(* Logix 5000 project; controller LeakTestAuto vendor 1 type 14 code 226 rev 37.11; software revision 37.01; part 2 of 14 *)

ADD_ON_INSTRUCTION AOI_RobotPositions   (* revision 1.0 *)
VAR_OUTPUT
   LoadingNest : DINT; {access Read Only}
   Barcode : DINT; {access Read Only}
   TestingNest1 : DINT; {access Read Only}
   TestingNest2 : DINT; {access Read Only}
   PassChute : DINT; {access Read Only}
   FailChute : DINT; {access Read Only}
END_VAR

ROUTINE Logic   (* structured text *)
   LoadingNest := 0;
   Barcode := 1;
   TestingNest1 := 2;
   TestingNest2 := 3;
   PassChute := 4;
   FailChute := 5;
END_ROUTINE
END_ADD_ON_INSTRUCTION

ADD_ON_INSTRUCTION AOI_Sequencer_x64   (* revision 1.0 *)
VAR_IN_OUT
   SequenceStructure : udt_SequenceStructure_X64; {required}
END_VAR
VAR_INPUT
   inpNextStepInterlock : BOOL; {access Read Only, required}
   inpCyclePause : BOOL; {access Read Only, required}
   inpStepMode : BOOL; {access Read Only, required}
END_VAR
VAR
   FFLUDumpREAL : REAL; {access None}
   Seq_FFLU_Cycle : CONTROL := (LEN := 10); {access None}
   Seq_FFLU_Step : CONTROL := (LEN := 64); {access None}
   Seq_FFLU_StepHist : CONTROL := (LEN := 64); {access None}
   FFLUDumpINT : INT; {access None}
   AvgContol : CONTROL := (LEN := 10); {access None}
END_VAR

ROUTINE Logic   (* ladder *)
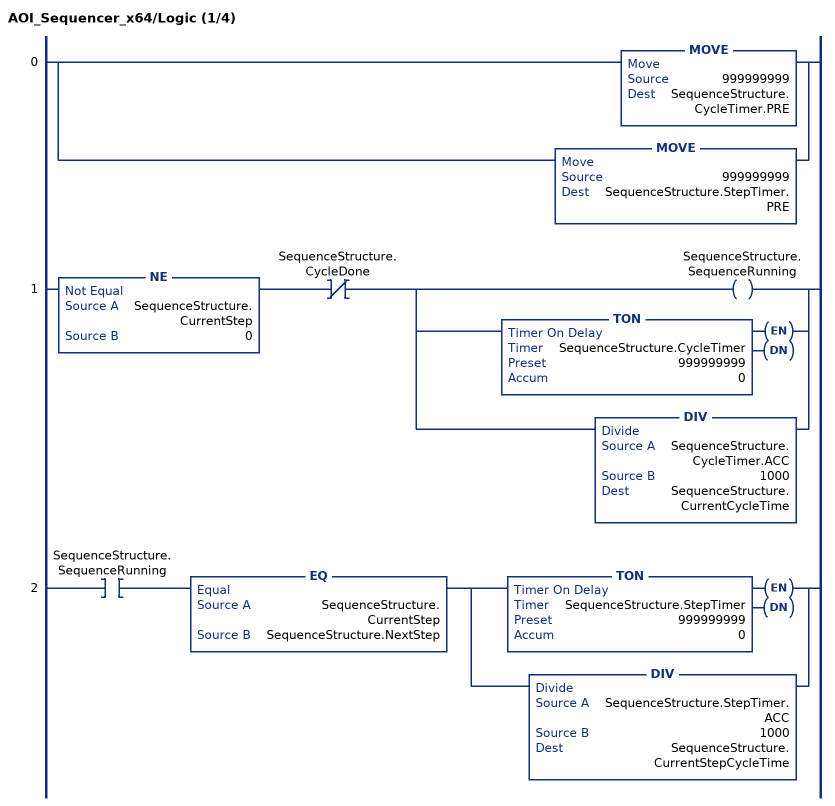
   0: [MOVE(999999999,SequenceStructure.CycleTimer.PRE) ,MOVE(999999999,SequenceStructure.StepTimer.PRE) ];
   1: NE(SequenceStructure.CurrentStep,0)XIO(SequenceStructure.CycleDone)[OTE(SequenceStructure.SequenceRunning) ,TON(SequenceStructure.CycleTimer,999999999,0) ,DIV(SequenceStructure.CycleTimer.ACC,1000,SequenceStructure.CurrentCycleTime) ];
   2: XIC(SequenceStructure.SequenceRunning)EQ(SequenceStructure.CurrentStep,SequenceStructure.NextStep)[TON(SequenceStructure.StepTimer,999999999,0) ,DIV(SequenceStructure.StepTimer.ACC,1000,SequenceStructure.CurrentStepCycleTime) ];
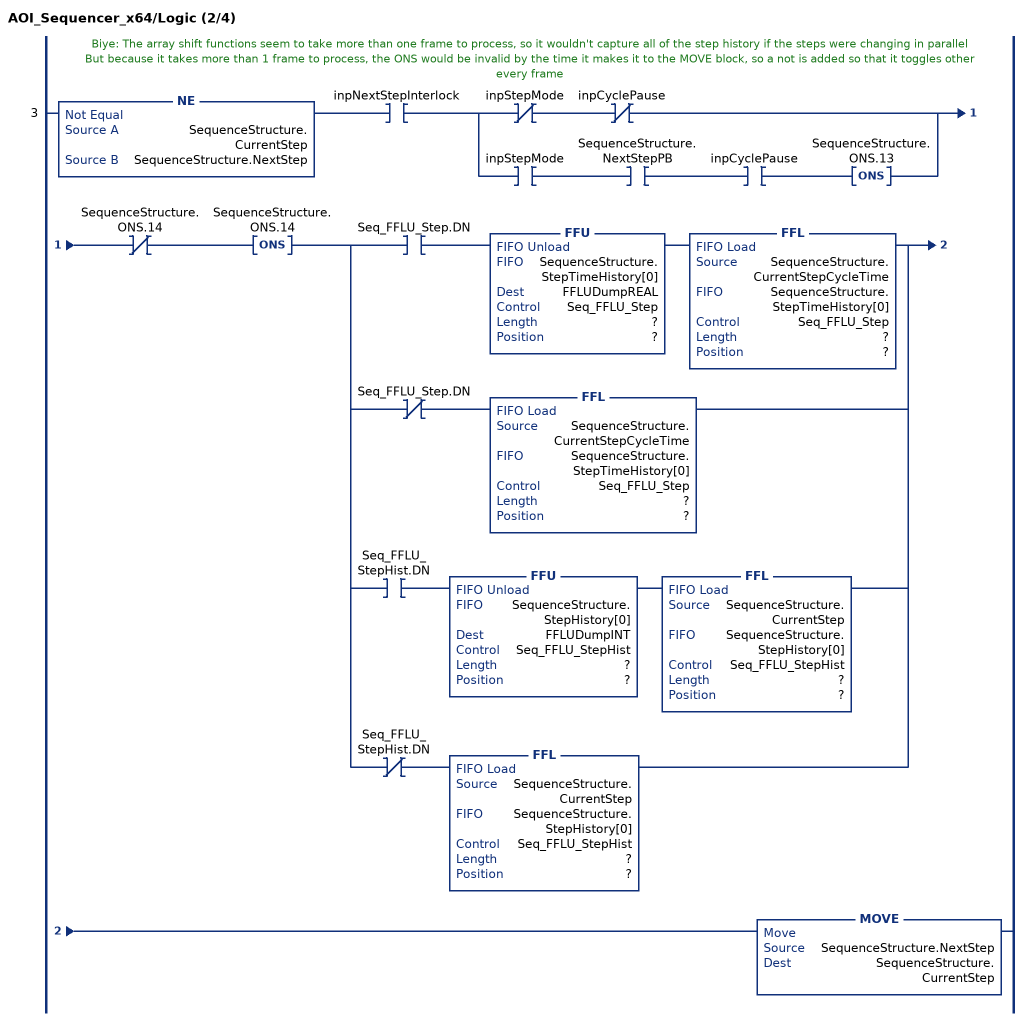
   // Biye: The array shift functions seem to take more than one frame to process, so it wouldn't capture all of the step history if the steps were changing in parallel
   // But because it takes more than 1 frame to process, the ONS would be invalid by the time it makes it to the MOVE block, so a not is added so that it toggles other every frame
   3: NE(SequenceStructure.CurrentStep,SequenceStructure.NextStep)XIC(inpNextStepInterlock)[XIO(inpStepMode) XIO(inpCyclePause) ,XIC(inpStepMode) XIC(SequenceStructure.NextStepPB) XIC(inpCyclePause) ONS(SequenceStructure.ONS.13) ]XIO(SequenceStructure.ONS.14)ONS(SequenceStructure.ONS.14)[XIC(Seq_FFLU_Step.DN) FFU(SequenceStructure.StepTimeHistory[0],FFLUDumpREAL,Seq_FFLU_Step,?,?) FFL(SequenceStructure.CurrentStepCycleTime,SequenceStructure.StepTimeHistory[0],Seq_FFLU_Step,?,?) ,XIO(Seq_FFLU_Step.DN) FFL(SequenceStructure.CurrentStepCycleTime,SequenceStructure.StepTimeHistory[0],Seq_FFLU_Step,?,?) ,XIC(Seq_FFLU_StepHist.DN) FFU(SequenceStructure.StepHistory[0],FFLUDumpINT,Seq_FFLU_StepHist,?,?) FFL(SequenceStructure.CurrentStep,SequenceStructure.StepHistory[0],Seq_FFLU_StepHist,?,?) ,XIO(Seq_FFLU_StepHist.DN) FFL(SequenceStructure.CurrentStep,SequenceStructure.StepHistory[0],Seq_FFLU_StepHist,?,?) ]MOVE(SequenceStructure.NextStep,SequenceStructure.CurrentStep);
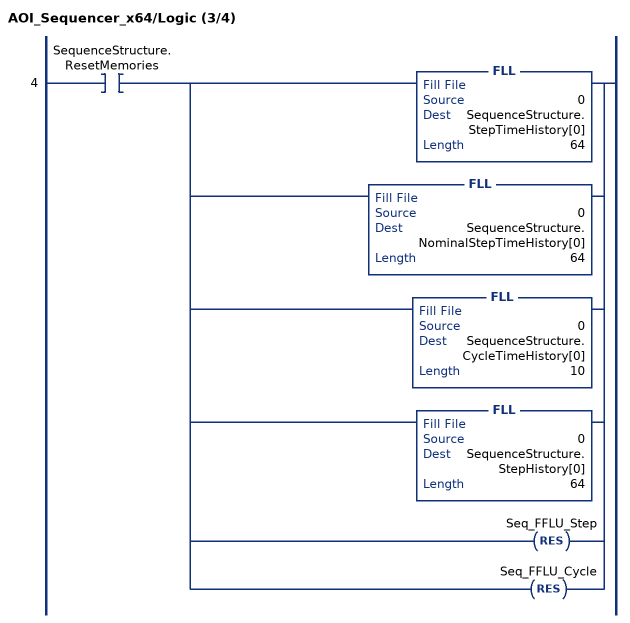
   4: XIC(SequenceStructure.ResetMemories)[FLL(0,SequenceStructure.StepTimeHistory[0],64) ,FLL(0,SequenceStructure.NominalStepTimeHistory[0],64) ,FLL(0,SequenceStructure.CycleTimeHistory[0],10) ,FLL(0,SequenceStructure.StepHistory[0],64) ,RES(Seq_FFLU_Step) ,RES(Seq_FFLU_Cycle) ];
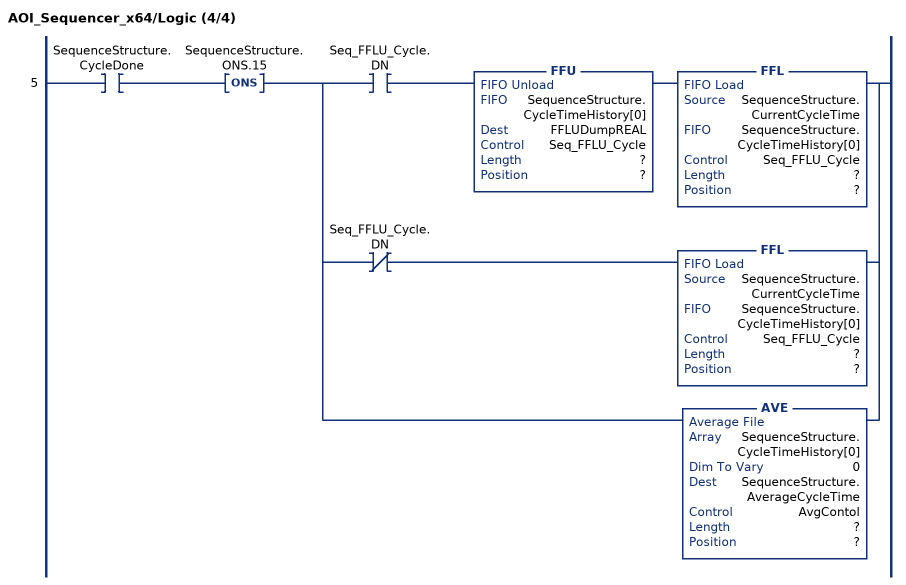
   5: XIC(SequenceStructure.CycleDone)ONS(SequenceStructure.ONS.15)[XIC(Seq_FFLU_Cycle.DN) FFU(SequenceStructure.CycleTimeHistory[0],FFLUDumpREAL,Seq_FFLU_Cycle,?,?) FFL(SequenceStructure.CurrentCycleTime,SequenceStructure.CycleTimeHistory[0],Seq_FFLU_Cycle,?,?) ,XIO(Seq_FFLU_Cycle.DN) FFL(SequenceStructure.CurrentCycleTime,SequenceStructure.CycleTimeHistory[0],Seq_FFLU_Cycle,?,?) ,AVE(SequenceStructure.CycleTimeHistory[0],0,SequenceStructure.AverageCycleTime,AvgContol,?,?) ];
END_ROUTINE
END_ADD_ON_INSTRUCTION

ADD_ON_INSTRUCTION AOI_StandardSeqSteps   (* revision 1.0 *)
VAR_OUTPUT
   Start : DINT; {access Read Only}
   ResultProcessing : DINT; {access Read Only}
   Complete : DINT; {access Read Only}
END_VAR

ROUTINE Logic   (* structured text *)
   Start := 1000;
   ResultProcessing := 8000;
   Complete := 9000;
END_ROUTINE
END_ADD_ON_INSTRUCTION

VAR_GLOBAL   (* controller tags *)
   AOI_IOCounter : AOI_IOCounter;
   ConveyorPurgeCounter : DINT;   // Outfeed Coveyor Purge Counter
   DateString : String20 := '07/14/2026';
   DateTimeString : String20 := '07/14/2026 13:25:59';
   Delay_TMR : TIMER[11] := ([0].PRE := 500, [1].PRE := 500, [3].PRE := 1000, [10].PRE := 100);   // Delay Timers
   HMI_ClearProcessFaultCounts_PB : BOOL;
   HMI_PurgeCycleSP : DINT := 20;   // HMI Purge Cycles Setpoint
   I_OP220_N3_CONVEYOR_CLEAT : ALIAS FOR Local:3:I.Pt13.Data;
   I_OP220_N3_CONVEYOR_LOAD : ALIAS FOR Local:3:I.Pt12.Data;
   I_OP220_N3_CONVEYOR_UNLOAD : ALIAS FOR Local:3:I.Pt14.Data;
   I_OP220_N3_DUT_PRE_NEST_0 : ALIAS FOR Local:3:I.Pt00.Data;
   I_OP220_N3_DUT_PRE_NEST_1 : ALIAS FOR Local:3:I.Pt01.Data;
   I_OP220_N3_DUT_PRE_NEST_2 : ALIAS FOR Local:3:I.Pt02.Data;
   I_OP220_N3_MAIN_AIR_OK : ALIAS FOR Local:3:I.Pt07.Data;
   I_OP220_N3_NEST1_EXTEND : ALIAS FOR Local:3:I.Pt04.Data;
   I_OP220_N3_NEST1_HOME : ALIAS FOR Local:3:I.Pt03.Data;
   I_OP220_N3_NEST2_EXTEND : ALIAS FOR Local:3:I.Pt06.Data;
   I_OP220_N3_NEST2_HOME : ALIAS FOR Local:3:I.Pt05.Data;
   I_OP220_N3_REJECT_BIN_OK : ALIAS FOR Local:3:I.Pt09.Data;
   I_OP220_N3_REJECT_CHUTE_PART : ALIAS FOR Local:3:I.Pt10.Data;
   I_OP220_N4_AC_SURGE_OK : ALIAS FOR Local:4:I.Pt00.Data;
   I_OP220_N4_CONVEYOR_ALARM_OK : ALIAS FOR Local:4:I.Pt03.Data;
   I_OP220_N4_CONVEYOR_SPEED : ALIAS FOR Local:4:I.Pt02.Data;
   I_OP220_N4_DC_OK : ALIAS FOR Local:4:I.Pt01.Data;
   I_OP220_N4_DC_OK_PS2 : ALIAS FOR Local:4:I.Pt04.Data;
   Ignition_Bypass : BOOL := 1;
   Ignition_DataReady : BOOL;
   Ignition_DataReceived : BOOL;
   IOCounterHasRef : BOOL := 1;
   IOCounterLastData : INT[8] := ([0] := 30383, [1] := 27, [2] := -31920);
   IOLabels : STRING[128] := ([0] := 'SI_OP220_N1_LASER_AREA_NC12', [1] := 'SI_OP220_N1_LASER_GUARD_NC12', [3] := 'SI_OP220_N1_SSR_12', [4] := 'SI_OP220_N1_CTRL_VLAVE_NC1', [8] := 'SO_OP220_N2_SSR_1', [9] := 'SO_OP220_N2_SSR_2', [16] := 'I_OP220_N3_DUT_PRE_NEST_0', [17] := 'I_OP220_N3_DUT_PRE_NEST_1', [18] := 'I_OP220_N3_DUT_PRE_NEST_2', [19] := 'I_OP220_N3_NEST1_HOME', [20] := 'I_OP220_N3_NEST1_EXTEND', [21] := 'I_OP220_N3_NEST2_HOME', [22] := 'I_OP220_N3_NEST2_EXTEND', [23] := 'I_OP220_N3_MAIN_AIR_OK', [25] := 'I_OP220_N3_REJECT_BIN_OK', [26] := 'I_OP220_N3_REJECT_CHUTE_PART', [28] := 'I_OP220_N3_CONVEYOR_LOAD', [29] := 'I_OP220_N3_CONVEYOR_CLEAT', [30] := 'I_OP220_N3_CONVEYOR_UNLOAD', [32] := 'I_OP220_N4_AC_SURGE_OK', [33] := 'I_OP220_N4_DC_OK', [34] := 'I_OP220_N4_CONVEYOR_SPEED', [35] := 'I_OP220_N4_CONVEYOR_ALARM_OK', [36] := 'I_OP220_N4_DC_OK_PS2', [48] := 'O_OP220_N5_EN_LT_GN', [49] := 'O_OP220_N5_EN_LT_YE', [50] := 'O_OP220_N5_EN_LT_RD', [51] := 'O_OP220_N5_EN_LT_BU', [52] := 'O_OP220_N5_EN_MAIN_AIR', [53] := 'O_OP220_N5_EN_NEST1_EXT', [54] := 'O_OP220_N5_EN_NEST1_HOME', [55] := 'O_OP220_N5_EN_NEST2_EXT', [56] := 'O_OP220_N5_EN_NEST2_HOME', [57] := 'O_OP220_N5_EN_ROBOT_LATCHOFF', [58] := 'O_OP220_N5_EN_CONV_ALM_RST', [59] := 'O_OP220_N5_CONV_REV', [60] := 'O_OP220_N5_CONV_FWD', [62] := 'O_OP220_N5_EN_GRIPPER_GRIP', [63] := 'O_OP220_N5_EN_GRIPPER_UNGRIP');
   IOResetArray : INT[8];
   IOTriggerCounts : UDINT[128] := ([0] := 204299, [1] := 372945, [2] := 289990, [3] := 273, [4] := 284, [5] := 267, [6] := 273, [7] := 59, [8] := 521, [9] := 265, [10] := 457, [11] := 1168, [12] := 461, [13] := 232, [14] := 218066, [16] := 969840, [17] := 969667, [18] := 22, [19] := 986, [21] := 84223, [22] := 84230, [23] := 72795, [24] := 72777, [25] := 484, [26] := 4412, [28] := 201946, [29] := 3, [30] := 359046, [31] := 359046);
   James_Dint : DINT := 27;   // James Test Word
   LastPLCEdit : String20 := '12/31/1997 20:30:57';
   LastPLCEditHistory : String20[20] := ([0] := '12/31/1997 20:30:57', [1] := '12/31/1997 20:25:04', [2] := '12/31/1997 20:25:02', [3] := '12/31/1997 20:23:56', [4] := '07/13/2026 19:08:25', [5] := '07/13/2026 19:08:18', [6] := '07/13/2026 19:08:11', [7] := '07/13/2026 19:08:03', [8] := '07/13/2026 19:07:56', [9] := '07/13/2026 19:07:30', [10] := '07/13/2026 19:07:23', [11] := '07/13/2026 19:07:15', [12] := '07/13/2026 19:07:07', [13] := '07/13/2026 19:06:54', [14] := '07/13/2026 18:39:24', [15] := '07/13/2026 18:31:47', [16] := '07/13/2026 18:28:19', [17] := '07/13/2026 18:25:40', [18] := '07/13/2026 18:21:57', [19] := '07/13/2026 18:19:53');
   NoData : AB:5000_DI16:I:0;
   null : STRING;
   O_OP220_N5_CONV_FWD : ALIAS FOR Local:5:O.Pt12.Data;
   O_OP220_N5_CONV_REV : ALIAS FOR Local:5:O.Pt11.Data;
   O_OP220_N5_EN_CONV_ALM_RST : ALIAS FOR Local:5:O.Pt10.Data;
   O_OP220_N5_EN_GRIPPER_GRIP : ALIAS FOR Local:5:O.Pt14.Data;
   O_OP220_N5_EN_GRIPPER_UNGRIP : ALIAS FOR Local:5:O.Pt15.Data;
   O_OP220_N5_EN_LT_BU : ALIAS FOR Local:5:O.Pt03.Data;
   O_OP220_N5_EN_LT_GN : ALIAS FOR Local:5:O.Pt00.Data;
   O_OP220_N5_EN_LT_RD : ALIAS FOR Local:5:O.Pt02.Data;
   O_OP220_N5_EN_LT_YE : ALIAS FOR Local:5:O.Pt01.Data;
   O_OP220_N5_EN_MAIN_AIR : ALIAS FOR Local:5:O.Pt04.Data;
   O_OP220_N5_EN_NEST1_EXT : ALIAS FOR Local:5:O.Pt05.Data;
   O_OP220_N5_EN_NEST1_HOME : ALIAS FOR Local:5:O.Pt06.Data;
   O_OP220_N5_EN_NEST2_EXT : ALIAS FOR Local:5:O.Pt07.Data;
   O_OP220_N5_EN_NEST2_HOME : ALIAS FOR Local:5:O.Pt08.Data;
   O_OP220_N5_EN_ROBOT_LATCHOFF : ALIAS FOR Local:5:O.Pt09.Data;
   Oneshot : DINT;   // Oneshots
   OP220_ConsumedFromMain : DINT[50] := ([0] := 2, [1] := 3);
   OP220_ConsumedFromMain_PurgeModeEn : BOOL;
   OP220_ConsumedFromMain_RobotPickupSafe : BOOL := 1;
   OP220_EStop_OK : BOOL := 1;
   OP220_EStopTest_DCS : DCI_STOP := (ChannelA := 1, ChannelB := 1, InputStatus := 1, RestartType := 1, ColdStartType := 1, DiscrepancyTime := 250, O1 := 1);
   OP220_Power : BOOL := 1;
   OP220_ProducedForMain : DINT[50] := ([0] := 3); {produced}
   PLC : AOI_PLC := (AlwaysOn := 1, FlasherSlow := 1, FlasherFast := 1, SlowFlashTime := 2000, MediumFlashTime := 1000, FastFlashTime := 500, Year := 2026, Day := 14, Month := 7, Hour := 13, Minute := 25, Second := 59, MicroSecond := 766719, DOY := 195, SetTimePB := 1);
   Produced_SetTime : udt_Produced_SetTime := (SetTime[0] := 2020, SetTime[1] := 5, SetTime[2] := 21, SetTime[3] := 15, SetTime[4] := 59, SetTime[5] := 15); {produced}
   Purge_Count_DN : BOOL;   // Purge Counter Completed
   ShiftChange : BOOL;
   ShiftNumber : SINT := 1;
   SI_OP220_N1_CTRL_VLAVE_NC1 : ALIAS FOR Local:1:I.Pt04.Data;
   SI_OP220_N1_LASER_AREA_NC12 : ALIAS FOR Local:1:I.Pt00.Data;
   SI_OP220_N1_LASER_GUARD_NC12 : ALIAS FOR Local:1:I.Pt01.Data;
   SI_OP220_N1_SSR_12 : ALIAS FOR Local:1:I.Pt03.Data;
   SO_OP220_N2_SSR_1 : ALIAS FOR Local:2:O.Pt00.Data;
   SO_OP220_N2_SSR_2 : ALIAS FOR Local:2:O.Pt01.Data;
   ST1_Ignition_DataReady : BOOL;
   ST1_Ignition_DataReady_Setup : BOOL;
   ST1_Ignition_DataReceived : BOOL;
   ST1_Ignition_SerialNum : STRING := 'B252620969';
   ST1_Ignition_Status : DINT := -10;
   ST2_Ignition_DataReady : BOOL;
   ST2_Ignition_DataReady_Setup : BOOL;
   ST2_Ignition_DataReceived : BOOL;
   ST2_Ignition_SerialNum : STRING;
   ST2_Ignition_Status : DINT := -10;
   TimeString : String20 := '13:25:59';
   TON_PLC_BootUp : TIMER := (PRE := 10000);
END_VAR

PROGRAM MainProgram   (* main routine MainRoutine *)
VAR
   AOI_Barcode_Comms : AOI_CommStatus := (Cmd := 1, stsConnecting := 1, stsRunning := 1, stsFaultCode := 516);
   AOI_CapActuators_Seq : AOI_Sequencer_x64 := (inpNextStepInterlock := 1);
   AOI_CapCTS_Seq : AOI_Sequencer_x64 := (inpNextStepInterlock := 1);
   AOI_CapCylinders_Seq : AOI_Sequencer_x64 := (inpNextStepInterlock := 1);
   AOI_CapFail_Seq : AOI_Sequencer_x64 := (inpNextStepInterlock := 1);
   AOI_CapPass_Seq : AOI_Sequencer_x64 := (inpNextStepInterlock := 1);
   AOI_CapRobot_Seq : AOI_Sequencer_x64 := (inpNextStepInterlock := 1);
   AOI_CapShuffle_Seq : AOI_Sequencer_x64 := (inpNextStepInterlock := 1);
   AOI_Conveyor_Seq : AOI_Sequencer_x64 := (inpNextStepInterlock := 1);
   AOI_CTS1 : AOI_CTS_INSTRUMENT := (Change_Program_Number := 3, UID_of_Desired_Results := 43055, Include_Detailed_Results := 1, Results_Error := 1, UID_Time := 1300);
   AOI_CTS1_Comms : AOI_CommStatus := (Cmd := 1, stsFaulted := 1, stsRunning := 1, stsFaultCode := 516);
   AOI_CTS1_Seq : AOI_Sequencer_x64 := (inpNextStepInterlock := 1);
   AOI_CTS2 : AOI_CTS_INSTRUMENT := (Change_Program_Number := 3, UID_of_Desired_Results := 42054, Include_Detailed_Results := 1, Results_Error := 1, UID_Time := 1300);
   AOI_CTS2_Comms : AOI_CommStatus := (Cmd := 1, stsFaulted := 1, stsRunning := 1, stsFaultCode := 516);
   AOI_CTS2_Seq : AOI_Sequencer_x64 := (inpNextStepInterlock := 1);
   AOI_GetShift : AOI_GetShift := (PLCHour := 13, ShiftNumber := 1);
   AOI_OP220_HomingSeq : AOI_Sequencer_x64;
   AOI_OP220_Seq : AOI_Sequencer_x64 := (inpNextStepInterlock := 1);
   AOI_Robot_Comms : AOI_CommStatus := (Cmd := 1, stsRunning := 1, stsFaultCode := 272);
   AOI_RobotPos : AOI_RobotPositions := (Barcode := 1, TestingNest1 := 2, TestingNest2 := 3, PassChute := 4, FailChute := 5);
   AOI_SeqSteps : AOI_StandardSeqSteps := (Start := 1000, ResultProcessing := 8000, Complete := 9000);
   AOI_SRX100 : AOI_KeyenceBarcode := (ReadSuccess := 1);
   Barcode_ResultData : STR_Barcode := 'B252620969';
   BarcodeBypass : BOOL;
   BarcodeInputs : udt_KeyenceScannerInputs;
   BarcodeOutputs : udt_KeyenceScannerOutputs;
   BarcodeScanner : udt_OutputStructure := (IL := 1);
   CapActuators_BarcodeBad : COUNTER := (PRE := 999999999, CU := 1);
   CapActuators_BarcodeGood : COUNTER := (PRE := 999999999, ACC := 111, CU := 1);
   CapActuators_CTS1Bad : COUNTER := (PRE := 999999999, CU := 1);
   CapActuators_CTS1Good : COUNTER := (PRE := 999999999, ACC := 10, CU := 1);
   CapActuators_CTS2Bad : COUNTER := (PRE := 999999999, CU := 1);
   CapActuators_CTS2Good : COUNTER := (PRE := 999999999, ACC := 3, CU := 1);
   CapActuators_Nest1HasPart : BOOL := 1;
   CapActuators_Nest2HasPart : BOOL;
   CapActuators_Seq : udt_SequenceStructure_X64 := (ONS := -7937, CurrentCycleTime := 409000.0, StepTimer.PRE := 999999999, CycleTimer.PRE := 999999999);
   CapCTS_CTS1Bad : COUNTER := (PRE := 999999999, ACC := 356, CU := 1);
   CapCTS_CTS1Good : COUNTER := (PRE := 999999999, ACC := 2730, CU := 1);
   CapCTS_CTS2Bad : COUNTER := (PRE := 999999999, ACC := 1, CU := 1);
   CapCTS_CTS2Good : COUNTER := (PRE := 999999999, ACC := 3085, CU := 1);
   CapCTS_Nest1HasPart : BOOL := 1;
   CapCTS_Nest2HasPart : BOOL := 1;
   CapCTS_Seq : udt_SequenceStructure_X64 := (ONS := -8132, StepHistory[0] := 2000, StepHistory[1] := 2010, StepHistory[2] := 2000, StepHistory[3] := 2010, StepHistory[4] := 2000, StepHistory[5] := 2010, StepHistory[6] := 2000, StepHistory[7] := 2010, StepHistory[8] := 2000, StepHistory[9] := 2010, StepHistory[10] := 2000, StepHistory[11] := 2010, StepHistory[12] := 2000, StepHistory[13] := 2010, StepHistory[14] := 2000, StepHistory[15] := 2010, StepHistory[16] := 2000, StepHistory[17] := 2010, StepHistory[18] := 2000, StepHistory[19] := 2010, StepHistory[20] := 2000, StepHistory[21] := 2010, StepHistory[22] := 2000, StepHistory[23] := 2010, StepHistory[24] := 2000, StepHistory[25] := 2010, StepHistory[26] := 2000, StepHistory[27] := 2010, StepHistory[28] := 2000, StepHistory[29] := 2010, StepHistory[30] := 2000, StepHistory[31] := 2010, StepHistory[32] := 2000, StepHistory[33] := 2010, StepHistory[34] := 2000, StepHistory[35] := 2010, StepHistory[36] := 2000, StepHistory[37] := 2010, StepHistory[38] := 2000, StepHistory[39] := 2010, StepHistory[40] := 2000, StepHistory[41] := 2010, StepHistory[42] := 2000, StepHistory[43] := 2010, StepHistory[44] := 2000, StepHistory[45] := 2010, StepHistory[46] := 2000, StepHistory[47] := 2010, StepHistory[48] := 2000, StepHistory[49] := 2010, StepHistory[50] := 2000, StepHistory[51] := 2010, StepHistory[52] := 2000, StepHistory[53] := 2010, StepHistory[54] := 2000, StepHistory[55] := 2010, StepHistory[56] := 2000, StepHistory[57] := 2010, StepHistory[58] := 2000,
        StepHistory[59] := 2010, StepHistory[60] := 2000, StepHistory[61] := 2010, StepHistory[62] := 2000, StepHistory[63] := 2010, CurrentCycleTime := 66060.766, CurrentStepCycleTime := 387.139, StepTimeHistory[0] := 0.035, StepTimeHistory[1] := 21.3, StepTimeHistory[2] := 0.04, StepTimeHistory[3] := 21.295, StepTimeHistory[4] := 0.035, StepTimeHistory[5] := 21.266, StepTimeHistory[6] := 0.034, StepTimeHistory[7] := 21.271, StepTimeHistory[8] := 0.033, StepTimeHistory[9] := 21.285, StepTimeHistory[10] := 0.041, StepTimeHistory[11] := 21.294, StepTimeHistory[12] := 0.052, StepTimeHistory[13] := 21.304, StepTimeHistory[14] := 0.035, StepTimeHistory[15] := 21.297, StepTimeHistory[16] := 0.036, StepTimeHistory[17] := 21.266, StepTimeHistory[18] := 0.039, StepTimeHistory[19] := 21.292, StepTimeHistory[20] := 0.04, StepTimeHistory[21] := 21.273, StepTimeHistory[22] := 0.035, StepTimeHistory[23] := 21.271, StepTimeHistory[24] := 0.051, StepTimeHistory[25] := 21.29, StepTimeHistory[26] := 0.036, StepTimeHistory[27] := 21.274, StepTimeHistory[28] := 0.041, StepTimeHistory[29] := 21.289, StepTimeHistory[30] := 0.036, StepTimeHistory[31] := 21.285, StepTimeHistory[32] := 0.039, StepTimeHistory[33] := 21.296, StepTimeHistory[34] := 0.05, StepTimeHistory[35] := 21.273, StepTimeHistory[36] := 0.057, StepTimeHistory[37] := 21.274, StepTimeHistory[38] := 0.034, StepTimeHistory[39] := 21.285, StepTimeHistory[40] := 0.05, StepTimeHistory[41] := 21.27, StepTimeHistory[42] := 0.036, StepTimeHistory[43] := 21.29, StepTimeHistory[44] := 0.035, StepTimeHistory[45] := 21.309, StepTimeHistory[46] := 0.051, StepTimeHistory[47] := 21.274, StepTimeHistory[48] := 0.037, StepTimeHistory[49] := 21.315, StepTimeHistory[50] := 0.044, StepTimeHistory[51] := 21.296, StepTimeHistory[52] := 0.035,
        StepTimeHistory[53] := 21.271, StepTimeHistory[54] := 0.034, StepTimeHistory[55] := 21.289, StepTimeHistory[56] := 0.045, StepTimeHistory[57] := 21.29, StepTimeHistory[58] := 0.034, StepTimeHistory[59] := 21.296, StepTimeHistory[60] := 0.035, StepTimeHistory[61] := 21.293, StepTimeHistory[62] := 0.069, StepTimeHistory[63] := 21.691, StepTimer.PRE := 999999999, CycleTimer.PRE := 999999999);
   CapCylinders_Seq : udt_SequenceStructure_X64 := (ONS := -8192);
   CapFail_Seq : udt_SequenceStructure_X64 := (ONS := -8192);
   CapPass_Seq : udt_SequenceStructure_X64 := (ONS := -8191);
   CapRobot_IsNest : BOOL;
   CapRobot_Seq : udt_SequenceStructure_X64 := (ONS := -8191, StepHistory[0] := 2070, StepHistory[1] := 2000, StepHistory[2] := 2010, StepHistory[3] := 2020, StepHistory[4] := 2030, StepHistory[5] := 2050, StepHistory[6] := 2060, StepHistory[7] := 2070, StepHistory[8] := 2000, StepHistory[9] := 2010, StepHistory[10] := 2020, StepHistory[11] := 2030, StepHistory[12] := 2040, StepHistory[13] := 2050, StepHistory[14] := 2060, StepHistory[15] := 2070, StepHistory[16] := 2000, StepHistory[17] := 2010, StepHistory[18] := 2020, StepHistory[19] := 2030, StepHistory[20] := 2040, StepHistory[21] := 2050, StepHistory[22] := 2060, StepHistory[23] := 2070, StepHistory[24] := 2000, StepHistory[25] := 2010, StepHistory[26] := 2020, StepHistory[27] := 2030, StepHistory[28] := 2050, StepHistory[29] := 2060, StepHistory[30] := 2070, StepHistory[31] := 2000, StepHistory[32] := 2010, StepHistory[33] := 2020, StepHistory[34] := 2030, StepHistory[35] := 2050, StepHistory[36] := 2060, StepHistory[37] := 2070, StepHistory[38] := 2000, StepHistory[39] := 2010, StepHistory[40] := 2020, StepHistory[41] := 2030, StepHistory[42] := 2040, StepHistory[43] := 2050, StepHistory[44] := 2060, StepHistory[45] := 2070, StepHistory[46] := 2000, StepHistory[47] := 2010, StepHistory[48] := 2020, StepHistory[49] := 2030, StepHistory[50] := 2040, StepHistory[51] := 2050, StepHistory[52] := 2060, StepHistory[53] := 2070, StepHistory[54] := 2000, StepHistory[55] := 2010, StepHistory[56] := 2020, StepHistory[57] := 2030, StepHistory[58] := 2050,
        StepHistory[59] := 2060, StepHistory[60] := 2070, StepHistory[61] := 2000, StepHistory[62] := 2010, StepHistory[63] := 2020, CurrentCycleTime := 1115.231, CurrentStepCycleTime := 0.264, StepTimeHistory[0] := 0.789, StepTimeHistory[1] := 0.038, StepTimeHistory[2] := 1.379, StepTimeHistory[3] := 0.038, StepTimeHistory[4] := 0.759, StepTimeHistory[5] := 0.039, StepTimeHistory[6] := 0.908, StepTimeHistory[7] := 0.908, StepTimeHistory[8] := 0.908, StepTimeHistory[9] := 0.097, StepTimeHistory[10] := 0.039, StepTimeHistory[11] := 0.899, StepTimeHistory[12] := 0.089, StepTimeHistory[13] := 0.028, StepTimeHistory[14] := 0.909, StepTimeHistory[15] := 0.909, StepTimeHistory[16] := 0.909, StepTimeHistory[17] := 0.087, StepTimeHistory[18] := 0.029, StepTimeHistory[19] := 1.589, StepTimeHistory[20] := 0.099, StepTimeHistory[21] := 0.039, StepTimeHistory[22] := 1.559, StepTimeHistory[23] := 1.559, StepTimeHistory[24] := 1.559, StepTimeHistory[25] := 0.097, StepTimeHistory[26] := 0.029, StepTimeHistory[27] := 1.398, StepTimeHistory[28] := 0.038, StepTimeHistory[29] := 1.468, StepTimeHistory[30] := 1.468, StepTimeHistory[31] := 1.468, StepTimeHistory[32] := 0.088, StepTimeHistory[33] := 0.028, StepTimeHistory[34] := 1.279, StepTimeHistory[35] := 0.039, StepTimeHistory[36] := 1.399, StepTimeHistory[37] := 1.399, StepTimeHistory[38] := 0.028, StepTimeHistory[39] := 0.769, StepTimeHistory[40] := 0.029, StepTimeHistory[41] := 0.758, StepTimeHistory[42] := 0.009, StepTimeHistory[43] := 0.039, StepTimeHistory[44] := 0.66, StepTimeHistory[45] := 0.66, StepTimeHistory[46] := 0.66, StepTimeHistory[47] := 0.66, StepTimeHistory[48] := 0.037, StepTimeHistory[49] := 1.209, StepTimeHistory[50] := 0.099, StepTimeHistory[51] := 0.028, StepTimeHistory[52] := 1.049,
        StepTimeHistory[53] := 1.049, StepTimeHistory[54] := 1.049, StepTimeHistory[55] := 1.049, StepTimeHistory[56] := 0.036, StepTimeHistory[57] := 0.898, StepTimeHistory[58] := 0.038, StepTimeHistory[59] := 0.849, StepTimeHistory[60] := 0.849, StepTimeHistory[61] := 0.849, StepTimeHistory[62] := 0.849, StepTimeHistory[63] := 0.026, StepTimer.PRE := 999999999, CycleTimer.PRE := 999999999);
   CapRobot_StartPos : DINT := 1;
   CapRobot_TargetPos : DINT := 5;
   CapShuffle_CTS1Bad : COUNTER := (PRE := 999999999, ACC := 4, CU := 1);
   CapShuffle_CTS1Good : COUNTER := (PRE := 999999999, CU := 1);
   CapShuffle_CTS2Bad : COUNTER := (PRE := 999999999, ACC := 3, CU := 1);
   CapShuffle_CTS2Good : COUNTER := (PRE := 999999999, CU := 1);
   CapShuffle_Seq : udt_SequenceStructure_X64 := (ONS := -8161, StepHistory[0] := 5440, StepHistory[1] := 5450, StepHistory[2] := 4000, StepHistory[3] := 4010, StepHistory[4] := 4020, StepHistory[5] := 5000, StepHistory[6] := 5600, StepHistory[7] := 5610, StepHistory[8] := 5620, StepHistory[9] := 5630, StepHistory[10] := 5640, StepHistory[11] := 5650, StepHistory[12] := 4000, StepHistory[13] := 4010, StepHistory[14] := 4020, StepHistory[15] := 4030, StepHistory[16] := 5000, StepHistory[17] := 5100, StepHistory[18] := 5110, StepHistory[19] := 5120, StepHistory[20] := 5130, StepHistory[21] := 5400, StepHistory[22] := 5410, StepHistory[23] := 5420, StepHistory[24] := 5430, StepHistory[25] := 5440, StepHistory[26] := 5450, StepHistory[27] := 4000, StepHistory[28] := 4010, StepHistory[29] := 4020, StepHistory[30] := 5000, StepHistory[31] := 5600, StepHistory[32] := 5610, StepHistory[33] := 5620, StepHistory[34] := 5630, StepHistory[35] := 5640, StepHistory[36] := 5650, StepHistory[37] := 4000, StepHistory[38] := 4010, StepHistory[39] := 4020, StepHistory[40] := 4030, StepHistory[41] := 5000, StepHistory[42] := 5100, StepHistory[43] := 5110, StepHistory[44] := 5120, StepHistory[45] := 5130, StepHistory[46] := 5400, StepHistory[47] := 5410, StepHistory[48] := 5420, StepHistory[49] := 5430, StepHistory[50] := 5440, StepHistory[51] := 5450, StepHistory[52] := 4000, StepHistory[53] := 4010, StepHistory[54] := 4020, StepHistory[55] := 5000, StepHistory[56] := 5600, StepHistory[57] := 5610, StepHistory[58] := 5620,
        StepHistory[59] := 5630, StepHistory[60] := 5640, StepHistory[61] := 5650, StepHistory[62] := 4000, StepHistory[63] := 4010, CurrentCycleTime := 91.095, CurrentStepCycleTime := 4.506, StepTimeHistory[0] := 0.039, StepTimeHistory[1] := 0.659, StepTimeHistory[2] := 6.164, StepTimeHistory[3] := 0.527, StepTimeHistory[4] := 0.527, StepTimeHistory[5] := 0.527, StepTimeHistory[6] := 0.034, StepTimeHistory[7] := 0.89, StepTimeHistory[8] := 0.039, StepTimeHistory[9] := 1.599, StepTimeHistory[10] := 0.039, StepTimeHistory[11] := 1.058, StepTimeHistory[12] := 1.058, StepTimeHistory[13] := 1.058, StepTimeHistory[14] := 6.022, StepTimeHistory[15] := 0.541, StepTimeHistory[16] := 0.541, StepTimeHistory[17] := 0.042, StepTimeHistory[18] := 0.748, StepTimeHistory[19] := 0.039, StepTimeHistory[20] := 5.023, StepTimeHistory[21] := 0.035, StepTimeHistory[22] := 1.599, StepTimeHistory[23] := 0.039, StepTimeHistory[24] := 1.489, StepTimeHistory[25] := 0.04, StepTimeHistory[26] := 0.659, StepTimeHistory[27] := 6.163, StepTimeHistory[28] := 0.524, StepTimeHistory[29] := 0.524, StepTimeHistory[30] := 0.524, StepTimeHistory[31] := 0.038, StepTimeHistory[32] := 0.859, StepTimeHistory[33] := 0.039, StepTimeHistory[34] := 1.599, StepTimeHistory[35] := 0.039, StepTimeHistory[36] := 1.049, StepTimeHistory[37] := 1.049, StepTimeHistory[38] := 1.049, StepTimeHistory[39] := 6.021, StepTimeHistory[40] := 0.533, StepTimeHistory[41] := 0.533, StepTimeHistory[42] := 0.04, StepTimeHistory[43] := 0.739, StepTimeHistory[44] := 0.039, StepTimeHistory[45] := 5.084, StepTimeHistory[46] := 0.024, StepTimeHistory[47] := 1.569, StepTimeHistory[48] := 0.029, StepTimeHistory[49] := 1.469, StepTimeHistory[50] := 0.029, StepTimeHistory[51] := 0.66, StepTimeHistory[52] := 6.163,
        StepTimeHistory[53] := 0.541, StepTimeHistory[54] := 0.541, StepTimeHistory[55] := 0.541, StepTimeHistory[56] := 0.021, StepTimeHistory[57] := 0.879, StepTimeHistory[58] := 0.039, StepTimeHistory[59] := 1.569, StepTimeHistory[60] := 0.029, StepTimeHistory[61] := 1.059, StepTimeHistory[62] := 1.059, StepTimeHistory[63] := 1.059, StepTimer.PRE := 999999999, CycleTimer.PRE := 999999999);
   Config_ConveyorHomeCounter : DINT;
   Config_ConveyorHomeCounterEnter : BOOL;
   Config_CylinderWaitTime : DINT := 500;
   Config_CylinderWaitTimeEnter : BOOL;
   Config_MaxFailCount : DINT := 10;
   Config_MaxFailCountEnter : BOOL;
   Conveyor : udt_OutputStructure := (IL := 1, BC := 1);
   Conveyor_Seq : udt_SequenceStructure_X64 := (CycleDone := 1, CurrentStep := 9000, NextStep := 9000, ONS := -32768, StepHistory[0] := 9000, StepHistory[1] := 1000, StepHistory[2] := 1010, StepHistory[3] := 9000, StepHistory[4] := 1000, StepHistory[5] := 1010, StepHistory[6] := 9000, StepHistory[7] := 1000, StepHistory[8] := 1010, StepHistory[9] := 9000, StepHistory[10] := 1000, StepHistory[11] := 1010, StepHistory[12] := 9000, StepHistory[13] := 1000, StepHistory[14] := 1010, StepHistory[15] := 9000, StepHistory[16] := 1000, StepHistory[17] := 1010, StepHistory[18] := 9000, StepHistory[19] := 1000, StepHistory[20] := 1010, StepHistory[21] := 9000, StepHistory[22] := 1000, StepHistory[23] := 1010, StepHistory[24] := 9000, StepHistory[25] := 1000, StepHistory[26] := 1010, StepHistory[27] := 9000, StepHistory[28] := 1000, StepHistory[29] := 1010, StepHistory[30] := 9000, StepHistory[31] := 1000, StepHistory[32] := 1010, StepHistory[33] := 9000, StepHistory[34] := 1000, StepHistory[35] := 1010, StepHistory[36] := 9000, StepHistory[37] := 1000, StepHistory[38] := 1010, StepHistory[39] := 9000, StepHistory[40] := 1000, StepHistory[41] := 1010, StepHistory[42] := 9000, StepHistory[43] := 1000, StepHistory[44] := 1010, StepHistory[45] := 9000, StepHistory[46] := 1000, StepHistory[47] := 1010, StepHistory[48] := 9000, StepHistory[49] := 1000, StepHistory[50] := 1010, StepHistory[51] := 9000, StepHistory[52] := 1000, StepHistory[53] := 1010, StepHistory[54] := 9000, StepHistory[55] := 1000,
        StepHistory[56] := 1010, StepHistory[57] := 9000, StepHistory[58] := 1000, StepHistory[59] := 1010, StepHistory[60] := 9000, StepHistory[62] := 1000, StepHistory[63] := 1010, StepDescriptionPointer := -30912, CurrentCycleTime := 2.555, AverageCycleTime := 2.2348, PreviousCycleTime := 2706.0, CycleTimeHistory[0] := 2.54, CycleTimeHistory[1] := 2.424, CycleTimeHistory[2] := 2.46, CycleTimeHistory[3] := 2.48, CycleTimeHistory[4] := 2.5, CycleTimeHistory[5] := 2.455, CycleTimeHistory[6] := 2.46, CycleTimeHistory[7] := 2.474, CycleTimeHistory[9] := 2.555, CurrentStepCycleTime := 2.398, StepTimeHistory[0] := 2.354, StepTimeHistory[1] := 0.128, StepTimeHistory[2] := 2.349, StepTimeHistory[3] := 2.349, StepTimeHistory[4] := 0.128, StepTimeHistory[5] := 2.384, StepTimeHistory[6] := 2.384, StepTimeHistory[7] := 0.125, StepTimeHistory[8] := 2.323, StepTimeHistory[9] := 2.323, StepTimeHistory[10] := 0.129, StepTimeHistory[11] := 2.359, StepTimeHistory[12] := 2.359, StepTimeHistory[13] := 0.124, StepTimeHistory[14] := 2.355, StepTimeHistory[15] := 2.355, StepTimeHistory[16] := 0.129, StepTimeHistory[17] := 2.338, StepTimeHistory[18] := 2.338, StepTimeHistory[19] := 0.126, StepTimeHistory[20] := 2.324, StepTimeHistory[21] := 2.324, StepTimeHistory[22] := 0.124, StepTimeHistory[23] := 2.354, StepTimeHistory[24] := 2.354, StepTimeHistory[25] := 0.13, StepTimeHistory[26] := 2.369, StepTimeHistory[27] := 2.369, StepTimeHistory[28] := 0.124, StepTimeHistory[29] := 2.349, StepTimeHistory[30] := 2.349, StepTimeHistory[31] := 0.129, StepTimeHistory[32] := 2.324, StepTimeHistory[33] := 2.324, StepTimeHistory[34] := 0.124, StepTimeHistory[35] := 2.324, StepTimeHistory[36] := 2.324, StepTimeHistory[37] := 0.119, StepTimeHistory[38] := 2.419,
        StepTimeHistory[39] := 2.419, StepTimeHistory[40] := 0.124, StepTimeHistory[41] := 2.299, StepTimeHistory[42] := 2.299, StepTimeHistory[43] := 0.129, StepTimeHistory[44] := 2.329, StepTimeHistory[45] := 2.329, StepTimeHistory[46] := 0.135, StepTimeHistory[47] := 2.344, StepTimeHistory[48] := 2.344, StepTimeHistory[49] := 0.124, StepTimeHistory[50] := 2.374, StepTimeHistory[51] := 2.374, StepTimeHistory[52] := 0.129, StepTimeHistory[53] := 2.324, StepTimeHistory[54] := 2.324, StepTimeHistory[55] := 0.124, StepTimeHistory[56] := 2.334, StepTimeHistory[57] := 2.334, StepTimeHistory[58] := 0.129, StepTimeHistory[59] := 2.344, StepTimeHistory[60] := 2.344, StepTimeHistory[61] := 2.344, StepTimeHistory[62] := 0.155, StepTimeHistory[63] := 2.398, StepTimer.PRE := 999999999, CycleTimer.PRE := 999999999);
   ConveyorCleatSensorFault : BOOL;
   ConveyorHasParts : BOOL;
   ConveyorHomeCounter : COUNTER := (DN := 1);
   CTS1_BarcodeWrite : STRING80;
   CTS1_BasicResult : MESSAGE;
        MessageParameters(ServiceCode := 16#000e, DestinationTag := CTS1_Result.Basic, ...)
   CTS1_DataRead : STRING80;
   CTS1_DetailResult : MESSAGE;
        MessageParameters(ServiceCode := 16#000e, DestinationTag := CTS1_Result.Detailed, ...)
   CTS1_Inputs : udt_CTS_INPUTS_FROM;
   CTS1_LastResultEval : STRING16;
   CTS1_LastTestUID : DINT := 43022;
   CTS1_NextTestUID : DINT := 43022;
   CTS1_NumTestsInSeq : SINT := 1;
   CTS1_Outputs : udt_CTS_OUTPUTS_TO := (change_program := 1, program_num := 3);
   CTS1_ReadMsg : MESSAGE;
        MessageParameters(ServiceCode := 16#000e, DestinationTag := CTS1_DataRead.DATA[0], ...)
   CTS1_Ready : DINT;
   CTS1_Result : udt_CTS_RESULT := (UID := 43055, Basic.unique_id := 43022, Basic.channel_num := 1, Basic.program_num := 1, Basic.evaluation_code := 2, Basic.test_port := 1, Basic.year := 26, Basic.month := 6, Basic.date := 5, Basic.hour := 10, Basic.minute := 56, Basic.second := 7, Basic.flags := 12, Basic.Num_tests := 1, Basic.test_elements.test_type := 69, Basic.test_elements.test_eval := 2, Basic.test_elements.num_elements := 4, Detailed.unique_id := 43022, Detailed.num_elements := 4, Detailed.Test_Type := 69, Detailed.element_data[0].Variable_code := 245, Detailed.element_data[0].prec_code := 2, Detailed.element_data[0].Unit_code := 165, Detailed.element_data[0].result_measurement := 1000.0, Detailed.element_data[1].Variable_code := 13, Detailed.element_data[1].prec_code := 3, Detailed.element_data[1].Unit_code := 12, Detailed.element_data[1].result_measurement := 0.0047218055, Detailed.element_data[2].Variable_code := 247, Detailed.element_data[2].prec_code := 3, Detailed.element_data[2].Unit_code := 12, Detailed.element_data[2].result_measurement := 5.095699, Detailed.element_data[3].Variable_code := 295, Detailed.element_data[3].prec_code := 3, Detailed.element_data[3].Unit_code := 12, Detailed.element_data[3].result_measurement := 5.096928);
   CTS1_ResultHistoryLeak : udt_CTS_RESULT[10] := ([0].UID := 42950, [0].Basic.unique_id := 42950, [0].Basic.channel_num := 1, [0].Basic.program_num := 2, [0].Basic.evaluation_code := 1, [0].Basic.test_port := 1, [0].Basic.year := 26, [0].Basic.month := 6, [0].Basic.date := 4, [0].Basic.hour := 14, [0].Basic.minute := 59, [0].Basic.second := 52, [0].Basic.flags := 12, [0].Basic.Num_tests := 1, [0].Basic.test_elements.test_type := 66, [0].Basic.test_elements.test_eval := 1, [0].Basic.test_elements.num_elements := 16, [0].Detailed.unique_id := 42950, [0].Detailed.num_elements := 16, [0].Detailed.Test_Type := 66, [0].Detailed.element_data[0].Variable_code := 61, [0].Detailed.element_data[0].prec_code := 2, [0].Detailed.element_data[0].Unit_code := 60, [0].Detailed.element_data[0].result_measurement := -0.003911555, [0].Detailed.element_data[1].Variable_code := 28, [0].Detailed.element_data[1].prec_code := 3, [0].Detailed.element_data[1].Unit_code := 41, [0].Detailed.element_data[1].result_measurement := -7.916242e-05, [0].Detailed.element_data[2].Variable_code := 13, [0].Detailed.element_data[2].prec_code := 3, [0].Detailed.element_data[2].Unit_code := 12, [0].Detailed.element_data[2].result_measurement := 5.2312574, [0].Detailed.element_data[3].Variable_code := 75, [0].Detailed.element_data[3].prec_code := 2, [0].Detailed.element_data[3].Unit_code := 60, [0].Detailed.element_data[4].Variable_code := 60, [0].Detailed.element_data[4].prec_code := 2, [0].Detailed.element_data[4].Unit_code := 60, [0].Detailed.element_data[4].result_measurement := -0.012293458, [0].Detailed.element_data[5].Variable_code := 56, [0].Detailed.element_data[5].prec_code := 3, [0].Detailed.element_data[5].Unit_code := 41, [0].Detailed.element_data[5].result_measurement := -0.00016763806, [0].Detailed.element_data[6].Variable_code := 55, [0].Detailed.element_data[6].prec_code := 3, [0].Detailed.element_data[6].Unit_code := 12, [0].Detailed.element_data[6].result_measurement := 5.2312574, [0].Detailed.element_data[7].Variable_code := 58, [0].Detailed.element_data[7].prec_code := 2, [0].Detailed.element_data[7].Unit_code := 60, [0].Detailed.element_data[7].result_measurement := -1.0002404, [0].Detailed.element_data[8].Variable_code := 59, [0].Detailed.element_data[8].prec_code := 2, [0].Detailed.element_data[8].Unit_code := 60, [0].Detailed.element_data[8].result_measurement := 1.0002404, [0].Detailed.element_data[9].Variable_code := 12, [0].Detailed.element_data[9].prec_code := 3, [0].Detailed.element_data[9].Unit_code := 12, [0].Detailed.element_data[9].result_measurement := 5.000001, [0].Detailed.element_data[10].Variable_code := 62,
        [0].Detailed.element_data[10].prec_code := 2, [0].Detailed.element_data[10].Unit_code := 60, [0].Detailed.element_data[10].result_measurement := 1.1298805, [0].Detailed.element_data[11].Variable_code := 21, [0].Detailed.element_data[11].prec_code := 3, [0].Detailed.element_data[11].Unit_code := 41, [0].Detailed.element_data[11].result_measurement := 4.656613e-06, [0].Detailed.element_data[12].Variable_code := 25, [0].Detailed.element_data[12].prec_code := 3, [0].Detailed.element_data[12].Unit_code := 41, [0].Detailed.element_data[12].result_measurement := 0.023245811, [0].Detailed.element_data[13].Variable_code := 216, [0].Detailed.element_data[13].prec_code := 3, [0].Detailed.element_data[13].Unit_code := 41, [0].Detailed.element_data[13].result_measurement := -3.7252903e-05, [0].Detailed.element_data[14].Variable_code := 218, [0].Detailed.element_data[14].prec_code := 3, [0].Detailed.element_data[14].Unit_code := 41, [0].Detailed.element_data[14].result_measurement := 0.011632219, [0].Detailed.element_data[15].Variable_code := 295, [0].Detailed.element_data[15].prec_code := 3, [0].Detailed.element_data[15].Unit_code := 12, [0].Detailed.element_data[15].result_measurement := 5.2330365, [1].UID := 42953, [1].Basic.unique_id := 42953, [1].Basic.channel_num := 1, [1].Basic.program_num := 2, [1].Basic.evaluation_code := 1, [1].Basic.test_port := 1, [1].Basic.year := 26, [1].Basic.month := 6, [1].Basic.date := 4, [1].Basic.hour := 15, [1].Basic.minute := 3, [1].Basic.second := 37, [1].Basic.flags := 12, [1].Basic.Num_tests := 1, [1].Basic.test_elements.test_type := 66, [1].Basic.test_elements.test_eval := 1, [1].Basic.test_elements.num_elements := 16, [1].Detailed.unique_id := 42953, [1].Detailed.num_elements := 16, [1].Detailed.Test_Type := 66, [1].Detailed.element_data[0].Variable_code := 61, [1].Detailed.element_data[0].prec_code := 2, [1].Detailed.element_data[0].Unit_code := 60, [1].Detailed.element_data[0].result_measurement := 0.0055879354, [1].Detailed.element_data[1].Variable_code := 28, [1].Detailed.element_data[1].prec_code := 3, [1].Detailed.element_data[1].Unit_code := 41, [1].Detailed.element_data[1].result_measurement := 0.00012572855, [1].Detailed.element_data[2].Variable_code := 13, [1].Detailed.element_data[2].prec_code := 3, [1].Detailed.element_data[2].Unit_code := 12, [1].Detailed.element_data[2].result_measurement := 5.2312155, [1].Detailed.element_data[3].Variable_code := 75, [1].Detailed.element_data[3].prec_code := 2, [1].Detailed.element_data[3].Unit_code := 60, [1].Detailed.element_data[4].Variable_code := 60, [1].Detailed.element_data[4].prec_code := 2,
        [1].Detailed.element_data[4].Unit_code := 60, [1].Detailed.element_data[4].result_measurement := 0.0044703484, [1].Detailed.element_data[5].Variable_code := 56, [1].Detailed.element_data[5].prec_code := 3, [1].Detailed.element_data[5].Unit_code := 41, [1].Detailed.element_data[5].result_measurement := 1.3969839e-05, [1].Detailed.element_data[6].Variable_code := 55, [1].Detailed.element_data[6].prec_code := 3, [1].Detailed.element_data[6].Unit_code := 12, [1].Detailed.element_data[6].result_measurement := 5.2312155, [1].Detailed.element_data[7].Variable_code := 58, [1].Detailed.element_data[7].prec_code := 2, [1].Detailed.element_data[7].Unit_code := 60, [1].Detailed.element_data[7].result_measurement := -1.0002404, [1].Detailed.element_data[8].Variable_code := 59, [1].Detailed.element_data[8].prec_code := 2, [1].Detailed.element_data[8].Unit_code := 60, [1].Detailed.element_data[8].result_measurement := 1.0002404, [1].Detailed.element_data[9].Variable_code := 12, [1].Detailed.element_data[9].prec_code := 3, [1].Detailed.element_data[9].Unit_code := 12, [1].Detailed.element_data[9].result_measurement := 5.000001, [1].Detailed.element_data[10].Variable_code := 62, [1].Detailed.element_data[10].prec_code := 2, [1].Detailed.element_data[10].Unit_code := 60, [1].Detailed.element_data[10].result_measurement := 1.1298805, [1].Detailed.element_data[11].Variable_code := 21, [1].Detailed.element_data[11].prec_code := 3, [1].Detailed.element_data[11].Unit_code := 41, [1].Detailed.element_data[11].result_measurement := 4.656613e-06, [1].Detailed.element_data[12].Variable_code := 25, [1].Detailed.element_data[12].prec_code := 3, [1].Detailed.element_data[12].Unit_code := 41, [1].Detailed.element_data[12].result_measurement := 0.023245811, [1].Detailed.element_data[13].Variable_code := 216, [1].Detailed.element_data[13].prec_code := 3, [1].Detailed.element_data[13].Unit_code := 41, [1].Detailed.element_data[13].result_measurement := -3.7252903e-05, [1].Detailed.element_data[14].Variable_code := 218, [1].Detailed.element_data[14].prec_code := 3, [1].Detailed.element_data[14].Unit_code := 41, [1].Detailed.element_data[14].result_measurement := 0.011632219, [1].Detailed.element_data[15].Variable_code := 295, [1].Detailed.element_data[15].prec_code := 3, [1].Detailed.element_data[15].Unit_code := 12, [1].Detailed.element_data[15].result_measurement := 5.2327847, [2].UID := 42956, [2].Basic.unique_id := 42956, [2].Basic.channel_num := 1, [2].Basic.program_num := 2, [2].Basic.evaluation_code := 1, [2].Basic.test_port := 1, [2].Basic.year := 26, [2].Basic.month := 6, [2].Basic.date := 4, [2].Basic.hour := 15, [2].Basic.minute := 7, [2].Basic.second := 3, [2].Basic.flags := 12, [2].Basic.Num_tests := 1,
        [2].Basic.test_elements.test_type := 66, [2].Basic.test_elements.test_eval := 1, [2].Basic.test_elements.num_elements := 16, [2].Detailed.unique_id := 42956, [2].Detailed.num_elements := 16, [2].Detailed.Test_Type := 66, [2].Detailed.element_data[0].Variable_code := 61, [2].Detailed.element_data[0].prec_code := 2, [2].Detailed.element_data[0].Unit_code := 60, [2].Detailed.element_data[0].result_measurement := 0.02514571, [2].Detailed.element_data[1].Variable_code := 28, [2].Detailed.element_data[1].prec_code := 3, [2].Detailed.element_data[1].Unit_code := 41, [2].Detailed.element_data[1].result_measurement := 0.00052619725, [2].Detailed.element_data[2].Variable_code := 13, [2].Detailed.element_data[2].prec_code := 3, [2].Detailed.element_data[2].Unit_code := 12, [2].Detailed.element_data[2].result_measurement := 5.231444, [2].Detailed.element_data[3].Variable_code := 75, [2].Detailed.element_data[3].prec_code := 2, [2].Detailed.element_data[3].Unit_code := 60, [2].Detailed.element_data[4].Variable_code := 60, [2].Detailed.element_data[4].prec_code := 2, [2].Detailed.element_data[4].Unit_code := 60, [2].Detailed.element_data[4].result_measurement := 0.020675361, [2].Detailed.element_data[5].Variable_code := 56, [2].Detailed.element_data[5].prec_code := 3, [2].Detailed.element_data[5].Unit_code := 41, [2].Detailed.element_data[5].result_measurement := 0.00017695129, [2].Detailed.element_data[6].Variable_code := 55, [2].Detailed.element_data[6].prec_code := 3, [2].Detailed.element_data[6].Unit_code := 12, [2].Detailed.element_data[6].result_measurement := 5.231444, [2].Detailed.element_data[7].Variable_code := 58, [2].Detailed.element_data[7].prec_code := 2, [2].Detailed.element_data[7].Unit_code := 60, [2].Detailed.element_data[7].result_measurement := -1.0002404, [2].Detailed.element_data[8].Variable_code := 59, [2].Detailed.element_data[8].prec_code := 2, [2].Detailed.element_data[8].Unit_code := 60, [2].Detailed.element_data[8].result_measurement := 1.0002404, [2].Detailed.element_data[9].Variable_code := 12, [2].Detailed.element_data[9].prec_code := 3, [2].Detailed.element_data[9].Unit_code := 12, [2].Detailed.element_data[9].result_measurement := 5.000001, [2].Detailed.element_data[10].Variable_code := 62, [2].Detailed.element_data[10].prec_code := 2, [2].Detailed.element_data[10].Unit_code := 60, [2].Detailed.element_data[10].result_measurement := 1.1298805, [2].Detailed.element_data[11].Variable_code := 21, [2].Detailed.element_data[11].prec_code := 3, [2].Detailed.element_data[11].Unit_code := 41, [2].Detailed.element_data[11].result_measurement := 4.656613e-06, [2].Detailed.element_data[12].Variable_code := 25, [2].Detailed.element_data[12].prec_code := 3, [2].Detailed.element_data[12].Unit_code := 41, [2].Detailed.element_data[12].result_measurement := 0.023245811, [2].Detailed.element_data[13].Variable_code := 216, [2].Detailed.element_data[13].prec_code := 3, [2].Detailed.element_data[13].Unit_code := 41,
        [2].Detailed.element_data[13].result_measurement := -3.7252903e-05, [2].Detailed.element_data[14].Variable_code := 218, [2].Detailed.element_data[14].prec_code := 3, [2].Detailed.element_data[14].Unit_code := 41, [2].Detailed.element_data[14].result_measurement := 0.011632219, [2].Detailed.element_data[15].Variable_code := 295, [2].Detailed.element_data[15].prec_code := 3, [2].Detailed.element_data[15].Unit_code := 12, [2].Detailed.element_data[15].result_measurement := 5.2328033, [3].UID := 42959, [3].Basic.unique_id := 42959, [3].Basic.channel_num := 1, [3].Basic.program_num := 2, [3].Basic.evaluation_code := 1, [3].Basic.test_port := 1, [3].Basic.year := 26, [3].Basic.month := 6, [3].Basic.date := 4, [3].Basic.hour := 15, [3].Basic.minute := 8, [3].Basic.second := 17, [3].Basic.flags := 12, [3].Basic.Num_tests := 1, [3].Basic.test_elements.test_type := 66, [3].Basic.test_elements.test_eval := 1, [3].Basic.test_elements.num_elements := 16, [3].Detailed.unique_id := 42959, [3].Detailed.num_elements := 16, [3].Detailed.Test_Type := 66, [3].Detailed.element_data[0].Variable_code := 61, [3].Detailed.element_data[0].prec_code := 2, [3].Detailed.element_data[0].Unit_code := 60, [3].Detailed.element_data[1].Variable_code := 28, [3].Detailed.element_data[1].prec_code := 3, [3].Detailed.element_data[1].Unit_code := 41, [3].Detailed.element_data[1].result_measurement := -4.656613e-06, [3].Detailed.element_data[2].Variable_code := 13, [3].Detailed.element_data[2].prec_code := 3, [3].Detailed.element_data[2].Unit_code := 12, [3].Detailed.element_data[2].result_measurement := 5.2301817, [3].Detailed.element_data[3].Variable_code := 75, [3].Detailed.element_data[3].prec_code := 2, [3].Detailed.element_data[3].Unit_code := 60, [3].Detailed.element_data[4].Variable_code := 60, [3].Detailed.element_data[4].prec_code := 2, [3].Detailed.element_data[4].Unit_code := 60, [3].Detailed.element_data[4].result_measurement := 0.0027939677, [3].Detailed.element_data[5].Variable_code := 56, [3].Detailed.element_data[5].prec_code := 3, [3].Detailed.element_data[5].Unit_code := 41, [3].Detailed.element_data[5].result_measurement := -4.656613e-06, [3].Detailed.element_data[6].Variable_code := 55, [3].Detailed.element_data[6].prec_code := 3, [3].Detailed.element_data[6].Unit_code := 12, [3].Detailed.element_data[6].result_measurement := 5.2301817, [3].Detailed.element_data[7].Variable_code := 58, [3].Detailed.element_data[7].prec_code := 2, [3].Detailed.element_data[7].Unit_code := 60, [3].Detailed.element_data[7].result_measurement := -1.0002404, [3].Detailed.element_data[8].Variable_code := 59,
        [3].Detailed.element_data[8].prec_code := 2, [3].Detailed.element_data[8].Unit_code := 60, [3].Detailed.element_data[8].result_measurement := 1.0002404, [3].Detailed.element_data[9].Variable_code := 12, [3].Detailed.element_data[9].prec_code := 3, [3].Detailed.element_data[9].Unit_code := 12, [3].Detailed.element_data[9].result_measurement := 5.000001, [3].Detailed.element_data[10].Variable_code := 62, [3].Detailed.element_data[10].prec_code := 2, [3].Detailed.element_data[10].Unit_code := 60, [3].Detailed.element_data[10].result_measurement := 1.1298805, [3].Detailed.element_data[11].Variable_code := 21, [3].Detailed.element_data[11].prec_code := 3, [3].Detailed.element_data[11].Unit_code := 41, [3].Detailed.element_data[11].result_measurement := 4.656613e-06, [3].Detailed.element_data[12].Variable_code := 25, [3].Detailed.element_data[12].prec_code := 3, [3].Detailed.element_data[12].Unit_code := 41, [3].Detailed.element_data[12].result_measurement := 0.023245811, [3].Detailed.element_data[13].Variable_code := 216, [3].Detailed.element_data[13].prec_code := 3, [3].Detailed.element_data[13].Unit_code := 41, [3].Detailed.element_data[13].result_measurement := -3.7252903e-05, [3].Detailed.element_data[14].Variable_code := 218, [3].Detailed.element_data[14].prec_code := 3, [3].Detailed.element_data[14].Unit_code := 41, [3].Detailed.element_data[14].result_measurement := 0.011632219, [3].Detailed.element_data[15].Variable_code := 295, [3].Detailed.element_data[15].prec_code := 3, [3].Detailed.element_data[15].Unit_code := 12, [3].Detailed.element_data[15].result_measurement := 5.23197, [4].UID := 42962, [4].Basic.unique_id := 42962, [4].Basic.channel_num := 1, [4].Basic.program_num := 2, [4].Basic.evaluation_code := 1, [4].Basic.test_port := 1, [4].Basic.year := 26, [4].Basic.month := 6, [4].Basic.date := 4, [4].Basic.hour := 15, [4].Basic.minute := 9, [4].Basic.second := 47, [4].Basic.flags := 12, [4].Basic.Num_tests := 1, [4].Basic.test_elements.test_type := 66, [4].Basic.test_elements.test_eval := 1, [4].Basic.test_elements.num_elements := 16, [4].Detailed.unique_id := 42962, [4].Detailed.num_elements := 16, [4].Detailed.Test_Type := 66, [4].Detailed.element_data[0].Variable_code := 61, [4].Detailed.element_data[0].prec_code := 2, [4].Detailed.element_data[0].Unit_code := 60, [4].Detailed.element_data[0].result_measurement := 0.022351742, [4].Detailed.element_data[1].Variable_code := 28, [4].Detailed.element_data[1].prec_code := 3, [4].Detailed.element_data[1].Unit_code := 41, [4].Detailed.element_data[1].result_measurement := 0.0004656613, [4].Detailed.element_data[2].Variable_code := 13,
        [4].Detailed.element_data[2].prec_code := 3, [4].Detailed.element_data[2].Unit_code := 12, [4].Detailed.element_data[2].result_measurement := 5.2300653, [4].Detailed.element_data[3].Variable_code := 75, [4].Detailed.element_data[3].prec_code := 2, [4].Detailed.element_data[3].Unit_code := 60, [4].Detailed.element_data[4].Variable_code := 60, [4].Detailed.element_data[4].prec_code := 2, [4].Detailed.element_data[4].Unit_code := 60, [4].Detailed.element_data[4].result_measurement := 0.022910535, [4].Detailed.element_data[5].Variable_code := 56, [4].Detailed.element_data[5].prec_code := 3, [4].Detailed.element_data[5].Unit_code := 41, [4].Detailed.element_data[5].result_measurement := 0.00020023435, [4].Detailed.element_data[6].Variable_code := 55, [4].Detailed.element_data[6].prec_code := 3, [4].Detailed.element_data[6].Unit_code := 12, [4].Detailed.element_data[6].result_measurement := 5.2300653, [4].Detailed.element_data[7].Variable_code := 58, [4].Detailed.element_data[7].prec_code := 2, [4].Detailed.element_data[7].Unit_code := 60, [4].Detailed.element_data[7].result_measurement := -1.0002404, [4].Detailed.element_data[8].Variable_code := 59, [4].Detailed.element_data[8].prec_code := 2, [4].Detailed.element_data[8].Unit_code := 60, [4].Detailed.element_data[8].result_measurement := 1.0002404, [4].Detailed.element_data[9].Variable_code := 12, [4].Detailed.element_data[9].prec_code := 3, [4].Detailed.element_data[9].Unit_code := 12, [4].Detailed.element_data[9].result_measurement := 5.000001, [4].Detailed.element_data[10].Variable_code := 62, [4].Detailed.element_data[10].prec_code := 2, [4].Detailed.element_data[10].Unit_code := 60, [4].Detailed.element_data[10].result_measurement := 1.1298805, [4].Detailed.element_data[11].Variable_code := 21, [4].Detailed.element_data[11].prec_code := 3, [4].Detailed.element_data[11].Unit_code := 41, [4].Detailed.element_data[11].result_measurement := 4.656613e-06, [4].Detailed.element_data[12].Variable_code := 25, [4].Detailed.element_data[12].prec_code := 3, [4].Detailed.element_data[12].Unit_code := 41, [4].Detailed.element_data[12].result_measurement := 0.023245811, [4].Detailed.element_data[13].Variable_code := 216, [4].Detailed.element_data[13].prec_code := 3, [4].Detailed.element_data[13].Unit_code := 41, [4].Detailed.element_data[13].result_measurement := -3.7252903e-05, [4].Detailed.element_data[14].Variable_code := 218, [4].Detailed.element_data[14].prec_code := 3, [4].Detailed.element_data[14].Unit_code := 41, [4].Detailed.element_data[14].result_measurement := 0.011632219, [4].Detailed.element_data[15].Variable_code := 295, [4].Detailed.element_data[15].prec_code := 3, [4].Detailed.element_data[15].Unit_code := 12, [4].Detailed.element_data[15].result_measurement := 5.231574, [5].UID := 43002, [5].Basic.unique_id := 43002, [5].Basic.channel_num := 1, [5].Basic.program_num := 2, [5].Basic.evaluation_code := 1, [5].Basic.test_port := 1,
        [5].Basic.year := 26, [5].Basic.month := 6, [5].Basic.date := 5, [5].Basic.hour := 10, [5].Basic.minute := 14, [5].Basic.second := 6, [5].Basic.flags := 12, [5].Basic.Num_tests := 1, [5].Basic.test_elements.test_type := 66, [5].Basic.test_elements.test_eval := 1, [5].Basic.test_elements.num_elements := 16, [5].Detailed.unique_id := 43002, [5].Detailed.num_elements := 16, [5].Detailed.Test_Type := 66, [5].Detailed.element_data[0].Variable_code := 61, [5].Detailed.element_data[0].prec_code := 2, [5].Detailed.element_data[0].Unit_code := 60, [5].Detailed.element_data[0].result_measurement := 0.007264316, [5].Detailed.element_data[1].Variable_code := 28, [5].Detailed.element_data[1].prec_code := 3, [5].Detailed.element_data[1].Unit_code := 41, [5].Detailed.element_data[1].result_measurement := 0.00016298145, [5].Detailed.element_data[2].Variable_code := 13, [5].Detailed.element_data[2].prec_code := 3, [5].Detailed.element_data[2].Unit_code := 12, [5].Detailed.element_data[2].result_measurement := 5.1514387, [5].Detailed.element_data[3].Variable_code := 75, [5].Detailed.element_data[3].prec_code := 2, [5].Detailed.element_data[3].Unit_code := 60, [5].Detailed.element_data[4].Variable_code := 60, [5].Detailed.element_data[4].prec_code := 2, [5].Detailed.element_data[4].Unit_code := 60, [5].Detailed.element_data[4].result_measurement := 0.0033527613, [5].Detailed.element_data[5].Variable_code := 56, [5].Detailed.element_data[5].prec_code := 3, [5].Detailed.element_data[5].Unit_code := 41, [5].Detailed.element_data[6].Variable_code := 55, [5].Detailed.element_data[6].prec_code := 3, [5].Detailed.element_data[6].Unit_code := 12, [5].Detailed.element_data[6].result_measurement := 5.1514387, [5].Detailed.element_data[7].Variable_code := 58, [5].Detailed.element_data[7].prec_code := 2, [5].Detailed.element_data[7].Unit_code := 60, [5].Detailed.element_data[7].result_measurement := -1.0002404, [5].Detailed.element_data[8].Variable_code := 59, [5].Detailed.element_data[8].prec_code := 2, [5].Detailed.element_data[8].Unit_code := 60, [5].Detailed.element_data[8].result_measurement := 1.0002404, [5].Detailed.element_data[9].Variable_code := 12, [5].Detailed.element_data[9].prec_code := 3, [5].Detailed.element_data[9].Unit_code := 12, [5].Detailed.element_data[9].result_measurement := 5.000001, [5].Detailed.element_data[10].Variable_code := 62, [5].Detailed.element_data[10].prec_code := 2, [5].Detailed.element_data[10].Unit_code := 60, [5].Detailed.element_data[10].result_measurement := 1.1298805, [5].Detailed.element_data[11].Variable_code := 21, [5].Detailed.element_data[11].prec_code := 3, [5].Detailed.element_data[11].Unit_code := 41, [5].Detailed.element_data[11].result_measurement := 4.656613e-06,
        [5].Detailed.element_data[12].Variable_code := 25, [5].Detailed.element_data[12].prec_code := 3, [5].Detailed.element_data[12].Unit_code := 41, [5].Detailed.element_data[12].result_measurement := 0.023245811, [5].Detailed.element_data[13].Variable_code := 216, [5].Detailed.element_data[13].prec_code := 3, [5].Detailed.element_data[13].Unit_code := 41, [5].Detailed.element_data[13].result_measurement := -3.7252903e-05, [5].Detailed.element_data[14].Variable_code := 218, [5].Detailed.element_data[14].prec_code := 3, [5].Detailed.element_data[14].Unit_code := 41, [5].Detailed.element_data[14].result_measurement := 0.011632219, [5].Detailed.element_data[15].Variable_code := 295, [5].Detailed.element_data[15].prec_code := 3, [5].Detailed.element_data[15].Unit_code := 12, [5].Detailed.element_data[15].result_measurement := 5.152752, [6].UID := 43008, [6].Basic.unique_id := 43008, [6].Basic.channel_num := 1, [6].Basic.program_num := 2, [6].Basic.evaluation_code := 1, [6].Basic.test_port := 1, [6].Basic.year := 26, [6].Basic.month := 6, [6].Basic.date := 5, [6].Basic.hour := 10, [6].Basic.minute := 17, [6].Basic.second := 58, [6].Basic.flags := 12, [6].Basic.Num_tests := 1, [6].Basic.test_elements.test_type := 66, [6].Basic.test_elements.test_eval := 1, [6].Basic.test_elements.num_elements := 16, [6].Detailed.unique_id := 43008, [6].Detailed.num_elements := 16, [6].Detailed.Test_Type := 66, [6].Detailed.element_data[0].Variable_code := 61, [6].Detailed.element_data[0].prec_code := 2, [6].Detailed.element_data[0].Unit_code := 60, [6].Detailed.element_data[0].result_measurement := 0.0067055225, [6].Detailed.element_data[1].Variable_code := 28, [6].Detailed.element_data[1].prec_code := 3, [6].Detailed.element_data[1].Unit_code := 41, [6].Detailed.element_data[1].result_measurement := 0.00014901161, [6].Detailed.element_data[2].Variable_code := 13, [6].Detailed.element_data[2].prec_code := 3, [6].Detailed.element_data[2].Unit_code := 12, [6].Detailed.element_data[2].result_measurement := 5.146321, [6].Detailed.element_data[3].Variable_code := 75, [6].Detailed.element_data[3].prec_code := 2, [6].Detailed.element_data[3].Unit_code := 60, [6].Detailed.element_data[4].Variable_code := 60, [6].Detailed.element_data[4].prec_code := 2, [6].Detailed.element_data[4].Unit_code := 60, [6].Detailed.element_data[4].result_measurement := 0.011734664, [6].Detailed.element_data[5].Variable_code := 56, [6].Detailed.element_data[5].prec_code := 3, [6].Detailed.element_data[5].Unit_code := 41, [6].Detailed.element_data[5].result_measurement := 8.8475645e-05, [6].Detailed.element_data[6].Variable_code := 55,
        [6].Detailed.element_data[6].prec_code := 3, [6].Detailed.element_data[6].Unit_code := 12, [6].Detailed.element_data[6].result_measurement := 5.146321, [6].Detailed.element_data[7].Variable_code := 58, [6].Detailed.element_data[7].prec_code := 2, [6].Detailed.element_data[7].Unit_code := 60, [6].Detailed.element_data[7].result_measurement := -1.0002404, [6].Detailed.element_data[8].Variable_code := 59, [6].Detailed.element_data[8].prec_code := 2, [6].Detailed.element_data[8].Unit_code := 60, [6].Detailed.element_data[8].result_measurement := 1.0002404, [6].Detailed.element_data[9].Variable_code := 12, [6].Detailed.element_data[9].prec_code := 3, [6].Detailed.element_data[9].Unit_code := 12, [6].Detailed.element_data[9].result_measurement := 5.000001, [6].Detailed.element_data[10].Variable_code := 62, [6].Detailed.element_data[10].prec_code := 2, [6].Detailed.element_data[10].Unit_code := 60, [6].Detailed.element_data[10].result_measurement := 1.1298805, [6].Detailed.element_data[11].Variable_code := 21, [6].Detailed.element_data[11].prec_code := 3, [6].Detailed.element_data[11].Unit_code := 41, [6].Detailed.element_data[11].result_measurement := 4.656613e-06, [6].Detailed.element_data[12].Variable_code := 25, [6].Detailed.element_data[12].prec_code := 3, [6].Detailed.element_data[12].Unit_code := 41, [6].Detailed.element_data[12].result_measurement := 0.023245811, [6].Detailed.element_data[13].Variable_code := 216, [6].Detailed.element_data[13].prec_code := 3, [6].Detailed.element_data[13].Unit_code := 41, [6].Detailed.element_data[13].result_measurement := -3.7252903e-05, [6].Detailed.element_data[14].Variable_code := 218, [6].Detailed.element_data[14].prec_code := 3, [6].Detailed.element_data[14].Unit_code := 41, [6].Detailed.element_data[14].result_measurement := 0.011632219, [6].Detailed.element_data[15].Variable_code := 295, [6].Detailed.element_data[15].prec_code := 3, [6].Detailed.element_data[15].Unit_code := 12, [6].Detailed.element_data[15].result_measurement := 5.1471496, [7].UID := 43011, [7].Basic.unique_id := 43011, [7].Basic.channel_num := 1, [7].Basic.program_num := 2, [7].Basic.evaluation_code := 1, [7].Basic.test_port := 1, [7].Basic.year := 26, [7].Basic.month := 6, [7].Basic.date := 5, [7].Basic.hour := 10, [7].Basic.minute := 18, [7].Basic.second := 57, [7].Basic.flags := 12, [7].Basic.Num_tests := 1, [7].Basic.test_elements.test_type := 66, [7].Basic.test_elements.test_eval := 1, [7].Basic.test_elements.num_elements := 16, [7].Detailed.unique_id := 43011, [7].Detailed.num_elements := 16, [7].Detailed.Test_Type := 66, [7].Detailed.element_data[0].Variable_code := 61,
        [7].Detailed.element_data[0].prec_code := 2, [7].Detailed.element_data[0].Unit_code := 60, [7].Detailed.element_data[0].result_measurement := -0.0033527613, [7].Detailed.element_data[1].Variable_code := 28, [7].Detailed.element_data[1].prec_code := 3, [7].Detailed.element_data[1].Unit_code := 41, [7].Detailed.element_data[1].result_measurement := -7.4505806e-05, [7].Detailed.element_data[2].Variable_code := 13, [7].Detailed.element_data[2].prec_code := 3, [7].Detailed.element_data[2].Unit_code := 12, [7].Detailed.element_data[2].result_measurement := 5.146088, [7].Detailed.element_data[3].Variable_code := 75, [7].Detailed.element_data[3].prec_code := 2, [7].Detailed.element_data[3].Unit_code := 60, [7].Detailed.element_data[4].Variable_code := 60, [7].Detailed.element_data[4].prec_code := 2, [7].Detailed.element_data[4].Unit_code := 60, [7].Detailed.element_data[4].result_measurement := 0.007264316, [7].Detailed.element_data[5].Variable_code := 56, [7].Detailed.element_data[5].prec_code := 3, [7].Detailed.element_data[5].Unit_code := 41, [7].Detailed.element_data[5].result_measurement := 4.1909516e-05, [7].Detailed.element_data[6].Variable_code := 55, [7].Detailed.element_data[6].prec_code := 3, [7].Detailed.element_data[6].Unit_code := 12, [7].Detailed.element_data[6].result_measurement := 5.146088, [7].Detailed.element_data[7].Variable_code := 58, [7].Detailed.element_data[7].prec_code := 2, [7].Detailed.element_data[7].Unit_code := 60, [7].Detailed.element_data[7].result_measurement := -1.0002404, [7].Detailed.element_data[8].Variable_code := 59, [7].Detailed.element_data[8].prec_code := 2, [7].Detailed.element_data[8].Unit_code := 60, [7].Detailed.element_data[8].result_measurement := 1.0002404, [7].Detailed.element_data[9].Variable_code := 12, [7].Detailed.element_data[9].prec_code := 3, [7].Detailed.element_data[9].Unit_code := 12, [7].Detailed.element_data[9].result_measurement := 5.000001, [7].Detailed.element_data[10].Variable_code := 62, [7].Detailed.element_data[10].prec_code := 2, [7].Detailed.element_data[10].Unit_code := 60, [7].Detailed.element_data[10].result_measurement := 1.1298805, [7].Detailed.element_data[11].Variable_code := 21, [7].Detailed.element_data[11].prec_code := 3, [7].Detailed.element_data[11].Unit_code := 41, [7].Detailed.element_data[11].result_measurement := 4.656613e-06, [7].Detailed.element_data[12].Variable_code := 25, [7].Detailed.element_data[12].prec_code := 3, [7].Detailed.element_data[12].Unit_code := 41, [7].Detailed.element_data[12].result_measurement := 0.023245811, [7].Detailed.element_data[13].Variable_code := 216, [7].Detailed.element_data[13].prec_code := 3, [7].Detailed.element_data[13].Unit_code := 41, [7].Detailed.element_data[13].result_measurement := -3.7252903e-05, [7].Detailed.element_data[14].Variable_code := 218, [7].Detailed.element_data[14].prec_code := 3, [7].Detailed.element_data[14].Unit_code := 41, [7].Detailed.element_data[14].result_measurement := 0.011632219, [7].Detailed.element_data[15].Variable_code := 295, [7].Detailed.element_data[15].prec_code := 3,
        [7].Detailed.element_data[15].Unit_code := 12, [7].Detailed.element_data[15].result_measurement := 5.147038, [8].UID := 43014, [8].Basic.unique_id := 43014, [8].Basic.channel_num := 1, [8].Basic.program_num := 2, [8].Basic.evaluation_code := 1, [8].Basic.test_port := 1, [8].Basic.year := 26, [8].Basic.month := 6, [8].Basic.date := 5, [8].Basic.hour := 10, [8].Basic.minute := 19, [8].Basic.second := 51, [8].Basic.flags := 12, [8].Basic.Num_tests := 1, [8].Basic.test_elements.test_type := 66, [8].Basic.test_elements.test_eval := 1, [8].Basic.test_elements.num_elements := 16, [8].Detailed.unique_id := 43014, [8].Detailed.num_elements := 16, [8].Detailed.Test_Type := 66, [8].Detailed.element_data[0].Variable_code := 61, [8].Detailed.element_data[0].prec_code := 2, [8].Detailed.element_data[0].Unit_code := 60, [8].Detailed.element_data[0].result_measurement := 0.007264316, [8].Detailed.element_data[1].Variable_code := 28, [8].Detailed.element_data[1].prec_code := 3, [8].Detailed.element_data[1].Unit_code := 41, [8].Detailed.element_data[1].result_measurement := 0.00015832484, [8].Detailed.element_data[2].Variable_code := 13, [8].Detailed.element_data[2].prec_code := 3, [8].Detailed.element_data[2].Unit_code := 12, [8].Detailed.element_data[2].result_measurement := 5.146228, [8].Detailed.element_data[3].Variable_code := 75, [8].Detailed.element_data[3].prec_code := 2, [8].Detailed.element_data[3].Unit_code := 60, [8].Detailed.element_data[4].Variable_code := 60, [8].Detailed.element_data[4].prec_code := 2, [8].Detailed.element_data[4].Unit_code := 60, [8].Detailed.element_data[4].result_measurement := 0.014528632, [8].Detailed.element_data[5].Variable_code := 56, [8].Detailed.element_data[5].prec_code := 3, [8].Detailed.element_data[5].Unit_code := 41, [8].Detailed.element_data[5].result_measurement := 0.00011641532, [8].Detailed.element_data[6].Variable_code := 55, [8].Detailed.element_data[6].prec_code := 3, [8].Detailed.element_data[6].Unit_code := 12, [8].Detailed.element_data[6].result_measurement := 5.146228, [8].Detailed.element_data[7].Variable_code := 58, [8].Detailed.element_data[7].prec_code := 2, [8].Detailed.element_data[7].Unit_code := 60, [8].Detailed.element_data[7].result_measurement := -1.0002404, [8].Detailed.element_data[8].Variable_code := 59, [8].Detailed.element_data[8].prec_code := 2, [8].Detailed.element_data[8].Unit_code := 60, [8].Detailed.element_data[8].result_measurement := 1.0002404, [8].Detailed.element_data[9].Variable_code := 12, [8].Detailed.element_data[9].prec_code := 3, [8].Detailed.element_data[9].Unit_code := 12,
        [8].Detailed.element_data[9].result_measurement := 5.000001, [8].Detailed.element_data[10].Variable_code := 62, [8].Detailed.element_data[10].prec_code := 2, [8].Detailed.element_data[10].Unit_code := 60, [8].Detailed.element_data[10].result_measurement := 1.1298805, [8].Detailed.element_data[11].Variable_code := 21, [8].Detailed.element_data[11].prec_code := 3, [8].Detailed.element_data[11].Unit_code := 41, [8].Detailed.element_data[11].result_measurement := 4.656613e-06, [8].Detailed.element_data[12].Variable_code := 25, [8].Detailed.element_data[12].prec_code := 3, [8].Detailed.element_data[12].Unit_code := 41, [8].Detailed.element_data[12].result_measurement := 0.023245811, [8].Detailed.element_data[13].Variable_code := 216, [8].Detailed.element_data[13].prec_code := 3, [8].Detailed.element_data[13].Unit_code := 41, [8].Detailed.element_data[13].result_measurement := -3.7252903e-05, [8].Detailed.element_data[14].Variable_code := 218, [8].Detailed.element_data[14].prec_code := 3, [8].Detailed.element_data[14].Unit_code := 41, [8].Detailed.element_data[14].result_measurement := 0.011632219, [8].Detailed.element_data[15].Variable_code := 295, [8].Detailed.element_data[15].prec_code := 3, [8].Detailed.element_data[15].Unit_code := 12, [8].Detailed.element_data[15].result_measurement := 5.14742);
   CTS1_ResultHistoryVol : udt_CTS_RESULT[10] := ([0].UID := 42958, [0].Basic.unique_id := 42958, [0].Basic.channel_num := 1, [0].Basic.program_num := 1, [0].Basic.evaluation_code := 1, [0].Basic.test_port := 1, [0].Basic.year := 26, [0].Basic.month := 6, [0].Basic.date := 4, [0].Basic.hour := 15, [0].Basic.minute := 8, [0].Basic.second := 10, [0].Basic.flags := 12, [0].Basic.Num_tests := 1, [0].Basic.test_elements.test_type := 69, [0].Basic.test_elements.test_eval := 1, [0].Basic.test_elements.num_elements := 4, [0].Detailed.unique_id := 42958, [0].Detailed.num_elements := 4, [0].Detailed.Test_Type := 69, [0].Detailed.element_data[0].Variable_code := 245, [0].Detailed.element_data[0].prec_code := 2, [0].Detailed.element_data[0].Unit_code := 165, [0].Detailed.element_data[0].result_measurement := 188.24182, [0].Detailed.element_data[1].Variable_code := 13, [0].Detailed.element_data[1].prec_code := 3, [0].Detailed.element_data[1].Unit_code := 12, [0].Detailed.element_data[1].result_measurement := 1.8080837, [0].Detailed.element_data[2].Variable_code := 247, [0].Detailed.element_data[2].prec_code := 3, [0].Detailed.element_data[2].Unit_code := 12, [0].Detailed.element_data[2].result_measurement := 5.211653, [0].Detailed.element_data[3].Variable_code := 295, [0].Detailed.element_data[3].prec_code := 3, [0].Detailed.element_data[3].Unit_code := 12, [0].Detailed.element_data[3].result_measurement := 5.2136693, [1].UID := 42961, [1].Basic.unique_id := 42961, [1].Basic.channel_num := 1, [1].Basic.program_num := 1, [1].Basic.evaluation_code := 1, [1].Basic.test_port := 1, [1].Basic.year := 26, [1].Basic.month := 6, [1].Basic.date := 4, [1].Basic.hour := 15, [1].Basic.minute := 9, [1].Basic.second := 40, [1].Basic.flags := 12, [1].Basic.Num_tests := 1, [1].Basic.test_elements.test_type := 69, [1].Basic.test_elements.test_eval := 1, [1].Basic.test_elements.num_elements := 4, [1].Detailed.unique_id := 42961, [1].Detailed.num_elements := 4, [1].Detailed.Test_Type := 69, [1].Detailed.element_data[0].Variable_code := 245, [1].Detailed.element_data[0].prec_code := 2, [1].Detailed.element_data[0].Unit_code := 165, [1].Detailed.element_data[0].result_measurement := 188.38309,
        [1].Detailed.element_data[1].Variable_code := 13, [1].Detailed.element_data[1].prec_code := 3, [1].Detailed.element_data[1].Unit_code := 12, [1].Detailed.element_data[1].result_measurement := 1.8068217, [1].Detailed.element_data[2].Variable_code := 247, [1].Detailed.element_data[2].prec_code := 3, [1].Detailed.element_data[2].Unit_code := 12, [1].Detailed.element_data[2].result_measurement := 5.2105684, [1].Detailed.element_data[3].Variable_code := 295, [1].Detailed.element_data[3].prec_code := 3, [1].Detailed.element_data[3].Unit_code := 12, [1].Detailed.element_data[3].result_measurement := 5.212333, [2].UID := 43001, [2].Basic.unique_id := 43001, [2].Basic.channel_num := 1, [2].Basic.program_num := 1, [2].Basic.evaluation_code := 1, [2].Basic.test_port := 1, [2].Basic.year := 26, [2].Basic.month := 6, [2].Basic.date := 5, [2].Basic.hour := 10, [2].Basic.minute := 13, [2].Basic.second := 59, [2].Basic.flags := 12, [2].Basic.Num_tests := 1, [2].Basic.test_elements.test_type := 69, [2].Basic.test_elements.test_eval := 1, [2].Basic.test_elements.num_elements := 4, [2].Detailed.unique_id := 43001, [2].Detailed.num_elements := 4, [2].Detailed.Test_Type := 69, [2].Detailed.element_data[0].Variable_code := 245, [2].Detailed.element_data[0].prec_code := 2, [2].Detailed.element_data[0].Unit_code := 165, [2].Detailed.element_data[0].result_measurement := 186.99532, [2].Detailed.element_data[1].Variable_code := 13, [2].Detailed.element_data[1].prec_code := 3, [2].Detailed.element_data[1].Unit_code := 12, [2].Detailed.element_data[1].result_measurement := 1.7807633, [2].Detailed.element_data[2].Variable_code := 247, [2].Detailed.element_data[2].prec_code := 3, [2].Detailed.element_data[2].Unit_code := 12, [2].Detailed.element_data[2].result_measurement := 5.1107073, [2].Detailed.element_data[3].Variable_code := 295, [2].Detailed.element_data[3].prec_code := 3, [2].Detailed.element_data[3].Unit_code := 12, [2].Detailed.element_data[3].result_measurement := 5.1116757, [3].UID := 43004, [3].Basic.unique_id := 43004, [3].Basic.channel_num := 1, [3].Basic.program_num := 1, [3].Basic.evaluation_code := 1, [3].Basic.test_port := 1, [3].Basic.year := 26, [3].Basic.month := 6, [3].Basic.date := 5, [3].Basic.hour := 10, [3].Basic.minute := 17, [3].Basic.second := 10,
        [3].Basic.flags := 12, [3].Basic.Num_tests := 1, [3].Basic.test_elements.test_type := 69, [3].Basic.test_elements.test_eval := 1, [3].Basic.test_elements.num_elements := 4, [3].Detailed.unique_id := 43004, [3].Detailed.num_elements := 4, [3].Detailed.Test_Type := 69, [3].Detailed.element_data[0].Variable_code := 245, [3].Detailed.element_data[0].prec_code := 2, [3].Detailed.element_data[0].Unit_code := 165, [3].Detailed.element_data[0].result_measurement := 187.00204, [3].Detailed.element_data[1].Variable_code := 13, [3].Detailed.element_data[1].prec_code := 3, [3].Detailed.element_data[1].Unit_code := 12, [3].Detailed.element_data[1].result_measurement := 1.779967, [3].Detailed.element_data[2].Variable_code := 247, [3].Detailed.element_data[2].prec_code := 3, [3].Detailed.element_data[2].Unit_code := 12, [3].Detailed.element_data[2].result_measurement := 5.108542, [3].Detailed.element_data[3].Variable_code := 295, [3].Detailed.element_data[3].prec_code := 3, [3].Detailed.element_data[3].Unit_code := 12, [3].Detailed.element_data[3].result_measurement := 5.1097245, [4].UID := 43007, [4].Basic.unique_id := 43007, [4].Basic.channel_num := 1, [4].Basic.program_num := 1, [4].Basic.evaluation_code := 1, [4].Basic.test_port := 1, [4].Basic.year := 26, [4].Basic.month := 6, [4].Basic.date := 5, [4].Basic.hour := 10, [4].Basic.minute := 17, [4].Basic.second := 51, [4].Basic.flags := 12, [4].Basic.Num_tests := 1, [4].Basic.test_elements.test_type := 69, [4].Basic.test_elements.test_eval := 1, [4].Basic.test_elements.num_elements := 4, [4].Detailed.unique_id := 43007, [4].Detailed.num_elements := 4, [4].Detailed.Test_Type := 69, [4].Detailed.element_data[0].Variable_code := 245, [4].Detailed.element_data[0].prec_code := 2, [4].Detailed.element_data[0].Unit_code := 165, [4].Detailed.element_data[0].result_measurement := 187.18288, [4].Detailed.element_data[1].Variable_code := 13, [4].Detailed.element_data[1].prec_code := 3, [4].Detailed.element_data[1].Unit_code := 12, [4].Detailed.element_data[1].result_measurement := 1.7796829, [4].Detailed.element_data[2].Variable_code := 247, [4].Detailed.element_data[2].prec_code := 3, [4].Detailed.element_data[2].Unit_code := 12, [4].Detailed.element_data[2].result_measurement := 5.1109447, [4].Detailed.element_data[3].Variable_code := 295, [4].Detailed.element_data[3].prec_code := 3, [4].Detailed.element_data[3].Unit_code := 12, [4].Detailed.element_data[3].result_measurement := 5.112132,
        [5].UID := 43010, [5].Basic.unique_id := 43010, [5].Basic.channel_num := 1, [5].Basic.program_num := 1, [5].Basic.evaluation_code := 1, [5].Basic.test_port := 1, [5].Basic.year := 26, [5].Basic.month := 6, [5].Basic.date := 5, [5].Basic.hour := 10, [5].Basic.minute := 18, [5].Basic.second := 50, [5].Basic.flags := 12, [5].Basic.Num_tests := 1, [5].Basic.test_elements.test_type := 69, [5].Basic.test_elements.test_eval := 1, [5].Basic.test_elements.num_elements := 4, [5].Detailed.unique_id := 43010, [5].Detailed.num_elements := 4, [5].Detailed.Test_Type := 69, [5].Detailed.element_data[0].Variable_code := 245, [5].Detailed.element_data[0].prec_code := 2, [5].Detailed.element_data[0].Unit_code := 165, [5].Detailed.element_data[0].result_measurement := 187.18771, [5].Detailed.element_data[1].Variable_code := 13, [5].Detailed.element_data[1].prec_code := 3, [5].Detailed.element_data[1].Unit_code := 12, [5].Detailed.element_data[1].result_measurement := 1.7792639, [5].Detailed.element_data[2].Variable_code := 247, [5].Detailed.element_data[2].prec_code := 3, [5].Detailed.element_data[2].Unit_code := 12, [5].Detailed.element_data[2].result_measurement := 5.109827, [5].Detailed.element_data[3].Variable_code := 295, [5].Detailed.element_data[3].prec_code := 3, [5].Detailed.element_data[3].Unit_code := 12, [5].Detailed.element_data[3].result_measurement := 5.1112704, [6].UID := 43013, [6].Basic.unique_id := 43013, [6].Basic.channel_num := 1, [6].Basic.program_num := 1, [6].Basic.evaluation_code := 1, [6].Basic.test_port := 1, [6].Basic.year := 26, [6].Basic.month := 6, [6].Basic.date := 5, [6].Basic.hour := 10, [6].Basic.minute := 19, [6].Basic.second := 44, [6].Basic.flags := 12, [6].Basic.Num_tests := 1, [6].Basic.test_elements.test_type := 69, [6].Basic.test_elements.test_eval := 1, [6].Basic.test_elements.num_elements := 4, [6].Detailed.unique_id := 43013, [6].Detailed.num_elements := 4, [6].Detailed.Test_Type := 69, [6].Detailed.element_data[0].Variable_code := 245, [6].Detailed.element_data[0].prec_code := 2, [6].Detailed.element_data[0].Unit_code := 165, [6].Detailed.element_data[0].result_measurement := 187.24707,
        [6].Detailed.element_data[1].Variable_code := 13, [6].Detailed.element_data[1].prec_code := 3, [6].Detailed.element_data[1].Unit_code := 12, [6].Detailed.element_data[1].result_measurement := 1.7789285, [6].Detailed.element_data[2].Variable_code := 247, [6].Detailed.element_data[2].prec_code := 3, [6].Detailed.element_data[2].Unit_code := 12, [6].Detailed.element_data[2].result_measurement := 5.10992, [6].Detailed.element_data[3].Variable_code := 295, [6].Detailed.element_data[3].prec_code := 3, [6].Detailed.element_data[3].Unit_code := 12, [6].Detailed.element_data[3].result_measurement := 5.111359, [7].UID := 43016, [7].Basic.unique_id := 43016, [7].Basic.channel_num := 1, [7].Basic.program_num := 1, [7].Basic.evaluation_code := 1, [7].Basic.test_port := 1, [7].Basic.year := 26, [7].Basic.month := 6, [7].Basic.date := 5, [7].Basic.hour := 10, [7].Basic.minute := 54, [7].Basic.second := 35, [7].Basic.flags := 12, [7].Basic.Num_tests := 1, [7].Basic.test_elements.test_type := 69, [7].Basic.test_elements.test_eval := 1, [7].Basic.test_elements.num_elements := 4, [7].Detailed.unique_id := 43016, [7].Detailed.num_elements := 4, [7].Detailed.Test_Type := 69, [7].Detailed.element_data[0].Variable_code := 245, [7].Detailed.element_data[0].prec_code := 2, [7].Detailed.element_data[0].Unit_code := 165, [7].Detailed.element_data[0].result_measurement := 187.26138, [7].Detailed.element_data[1].Variable_code := 13, [7].Detailed.element_data[1].prec_code := 3, [7].Detailed.element_data[1].Unit_code := 12, [7].Detailed.element_data[1].result_measurement := 1.7757015, [7].Detailed.element_data[2].Variable_code := 247, [7].Detailed.element_data[2].prec_code := 3, [7].Detailed.element_data[2].Unit_code := 12, [7].Detailed.element_data[2].result_measurement := 5.100905, [7].Detailed.element_data[3].Variable_code := 295, [7].Detailed.element_data[3].prec_code := 3, [7].Detailed.element_data[3].Unit_code := 12, [7].Detailed.element_data[3].result_measurement := 5.1019387, [8].UID := 43019, [8].Basic.unique_id := 43019, [8].Basic.channel_num := 1, [8].Basic.program_num := 1, [8].Basic.evaluation_code := 1, [8].Basic.test_port := 1, [8].Basic.year := 26, [8].Basic.month := 6, [8].Basic.date := 5, [8].Basic.hour := 10, [8].Basic.minute := 54, [8].Basic.second := 59,
        [8].Basic.flags := 12, [8].Basic.Num_tests := 1, [8].Basic.test_elements.test_type := 69, [8].Basic.test_elements.test_eval := 1, [8].Basic.test_elements.num_elements := 4, [8].Detailed.unique_id := 43019, [8].Detailed.num_elements := 4, [8].Detailed.Test_Type := 69, [8].Detailed.element_data[0].Variable_code := 245, [8].Detailed.element_data[0].prec_code := 2, [8].Detailed.element_data[0].Unit_code := 165, [8].Detailed.element_data[0].result_measurement := 187.70357, [8].Detailed.element_data[1].Variable_code := 13, [8].Detailed.element_data[1].prec_code := 3, [8].Detailed.element_data[1].Unit_code := 12, [8].Detailed.element_data[1].result_measurement := 1.7710496, [8].Detailed.element_data[2].Variable_code := 247, [8].Detailed.element_data[2].prec_code := 3, [8].Detailed.element_data[2].Unit_code := 12, [8].Detailed.element_data[2].result_measurement := 5.0953727, [8].Detailed.element_data[3].Variable_code := 295, [8].Detailed.element_data[3].prec_code := 3, [8].Detailed.element_data[3].Unit_code := 12, [8].Detailed.element_data[3].result_measurement := 5.096975, [9].UID := 43022, [9].Basic.unique_id := 43022, [9].Basic.channel_num := 1, [9].Basic.program_num := 1, [9].Basic.evaluation_code := 2, [9].Basic.test_port := 1, [9].Basic.year := 26, [9].Basic.month := 6, [9].Basic.date := 5, [9].Basic.hour := 10, [9].Basic.minute := 56, [9].Basic.second := 7, [9].Basic.flags := 12, [9].Basic.Num_tests := 1, [9].Basic.test_elements.test_type := 69, [9].Basic.test_elements.test_eval := 2, [9].Basic.test_elements.num_elements := 4, [9].Detailed.unique_id := 43022, [9].Detailed.num_elements := 4, [9].Detailed.Test_Type := 69, [9].Detailed.element_data[0].Variable_code := 245, [9].Detailed.element_data[0].prec_code := 2, [9].Detailed.element_data[0].Unit_code := 165, [9].Detailed.element_data[0].result_measurement := 1000.0, [9].Detailed.element_data[1].Variable_code := 13, [9].Detailed.element_data[1].prec_code := 3, [9].Detailed.element_data[1].Unit_code := 12, [9].Detailed.element_data[1].result_measurement := 0.0047218055, [9].Detailed.element_data[2].Variable_code := 247, [9].Detailed.element_data[2].prec_code := 3, [9].Detailed.element_data[2].Unit_code := 12, [9].Detailed.element_data[2].result_measurement := 5.095699, [9].Detailed.element_data[3].Variable_code := 295, [9].Detailed.element_data[3].prec_code := 3, [9].Detailed.element_data[3].Unit_code := 12, [9].Detailed.element_data[3].result_measurement := 5.096928);
   CTS1_Seq : udt_SequenceStructure_X64 := (CycleDone := 1, CurrentStep := 9000, NextStep := 9000, ONS := -32767, StepHistory[0] := 1000, StepHistory[1] := 1010, StepHistory[2] := 1020, StepHistory[3] := 1030, StepHistory[4] := 2000, StepHistory[5] := 2010, StepHistory[6] := 2020, StepHistory[7] := 2030, StepHistory[8] := 2000, StepHistory[9] := 2010, StepHistory[10] := 2020, StepHistory[11] := 2030, StepHistory[12] := 9000, StepHistory[13] := 1000, StepHistory[14] := 1010, StepHistory[15] := 1020, StepHistory[16] := 1030, StepHistory[17] := 2000, StepHistory[18] := 2010, StepHistory[19] := 2020, StepHistory[20] := 2030, StepHistory[21] := 2000, StepHistory[22] := 2010, StepHistory[23] := 2020, StepHistory[24] := 2030, StepHistory[25] := 9000, StepHistory[26] := 1000, StepHistory[27] := 1010, StepHistory[28] := 1020, StepHistory[29] := 1030, StepHistory[30] := 2000, StepHistory[31] := 2010, StepHistory[32] := 2020, StepHistory[33] := 2030, StepHistory[34] := 2000, StepHistory[35] := 2010, StepHistory[36] := 2020, StepHistory[37] := 2030, StepHistory[38] := 9000, StepHistory[39] := 1000, StepHistory[40] := 1010, StepHistory[41] := 1020, StepHistory[42] := 1030, StepHistory[43] := 2000, StepHistory[44] := 2010, StepHistory[45] := 2020, StepHistory[46] := 2030, StepHistory[47] := 2000, StepHistory[48] := 2010, StepHistory[49] := 2020, StepHistory[50] := 2030, StepHistory[51] := 9000, StepHistory[52] := 1000, StepHistory[53] := 1010, StepHistory[54] := 1020, StepHistory[55] := 1030,
        StepHistory[56] := 2000, StepHistory[57] := 2010, StepHistory[58] := 2020, StepHistory[59] := 2030, StepHistory[60] := 9000, StepHistory[61] := 1000, StepHistory[62] := 1010, StepHistory[63] := 1020, AverageCycleTime := 0.334, CycleTimeHistory[0] := 0.608, CycleTimeHistory[1] := 0.609, CycleTimeHistory[3] := 0.61, CycleTimeHistory[4] := 0.608, CycleTimeHistory[5] := 0.405, CycleTimeHistory[8] := 0.5, StepTimeHistory[1] := 0.199, StepTimeHistory[2] := 0.199, StepTimeHistory[3] := 0.199, StepTimeHistory[5] := 0.198, StepTimeHistory[6] := 0.198, StepTimeHistory[7] := 0.198, StepTimeHistory[9] := 0.199, StepTimeHistory[10] := 0.199, StepTimeHistory[11] := 0.199, StepTimeHistory[12] := 0.199, StepTimeHistory[14] := 0.199, StepTimeHistory[15] := 0.199, StepTimeHistory[16] := 0.199, StepTimeHistory[18] := 0.199, StepTimeHistory[19] := 0.199, StepTimeHistory[20] := 0.199, StepTimeHistory[22] := 0.2, StepTimeHistory[23] := 0.2, StepTimeHistory[24] := 0.2, StepTimeHistory[27] := 0.199, StepTimeHistory[28] := 0.199, StepTimeHistory[29] := 0.199, StepTimeHistory[31] := 0.2, StepTimeHistory[32] := 0.2, StepTimeHistory[33] := 0.2, StepTimeHistory[35] := 0.199, StepTimeHistory[36] := 0.199, StepTimeHistory[37] := 0.199, StepTimeHistory[38] := 0.199, StepTimeHistory[40] := 0.199, StepTimeHistory[41] := 0.199, StepTimeHistory[42] := 0.199, StepTimeHistory[44] := 0.199, StepTimeHistory[45] := 0.199, StepTimeHistory[46] := 0.199, StepTimeHistory[48] := 0.199, StepTimeHistory[49] := 0.199, StepTimeHistory[50] := 0.199, StepTimeHistory[51] := 0.199, StepTimeHistory[53] := 0.199, StepTimeHistory[54] := 0.199, StepTimeHistory[55] := 0.199, StepTimeHistory[57] := 0.2, StepTimeHistory[58] := 0.2, StepTimeHistory[59] := 0.2,
        StepTimeHistory[62] := 0.199, StepTimeHistory[63] := 0.299, StepTimer.PRE := 999999999, CycleTimer.PRE := 999999999);
   CTS1_SeqUID : DINT := 43055;
   CTS1_UIDMsg : MESSAGE;
        MessageParameters(ServiceCode := 16#0010, LocalElement := CTS1_Result.UID, ...)
   CTS1_WriteMsg : MESSAGE;
        MessageParameters(ServiceCode := 16#0010, LocalElement := CTS1_BarcodeWrite.DATA[0], ...)
   CTS2_BarcodeWrite : STRING80;
   CTS2_BasicResult : MESSAGE;
        MessageParameters(ServiceCode := 16#000e, DestinationTag := CTS2_Result.Basic, ...)
   CTS2_DataRead : STRING80;
   CTS2_DetailResult : MESSAGE;
        MessageParameters(ServiceCode := 16#000e, DestinationTag := CTS2_Result.Detailed, ...)
   CTS2_Inputs : udt_CTS_INPUTS_FROM;
   CTS2_LastResultEval : STRING16;
   CTS2_LastTestUID : DINT := 42024;
   CTS2_NextTestUID : DINT := 42024;
   CTS2_NumTestsInSeq : SINT := 2;
   CTS2_Outputs : udt_CTS_OUTPUTS_TO := (change_program := 1, program_num := 3);
   CTS2_ReadMsg : MESSAGE;
        MessageParameters(ServiceCode := 16#000e, DestinationTag := CTS2_DataRead.DATA[0], ...)
   CTS2_Ready : DINT;
   CTS2_Result : udt_CTS_RESULT := (UID := 42054, Basic.unique_id := 42024, Basic.channel_num := 1, Basic.program_num := 2, Basic.evaluation_code := 12, Basic.test_port := 1, Basic.year := 26, Basic.month := 6, Basic.date := 5, Basic.hour := 10, Basic.minute := 55, Basic.second := 45, Basic.flags := 12, Detailed.unique_id := 42024);
   CTS2_ResultHistoryLeak : udt_CTS_RESULT[10] := ([0].UID := 41949, [0].Basic.unique_id := 41949, [0].Basic.channel_num := 1, [0].Basic.program_num := 2, [0].Basic.evaluation_code := 1, [0].Basic.test_port := 1, [0].Basic.year := 26, [0].Basic.month := 6, [0].Basic.date := 4, [0].Basic.hour := 12, [0].Basic.minute := 28, [0].Basic.second := 18, [0].Basic.flags := 12, [0].Basic.Num_tests := 1, [0].Basic.test_elements.test_type := 66, [0].Basic.test_elements.test_eval := 1, [0].Basic.test_elements.num_elements := 16, [0].Detailed.unique_id := 41949, [0].Detailed.num_elements := 16, [0].Detailed.Test_Type := 66, [0].Detailed.element_data[0].Variable_code := 61, [0].Detailed.element_data[0].prec_code := 2, [0].Detailed.element_data[0].Unit_code := 60, [0].Detailed.element_data[0].result_measurement := -0.07376075, [0].Detailed.element_data[1].Variable_code := 28, [0].Detailed.element_data[1].prec_code := 3, [0].Detailed.element_data[1].Unit_code := 41, [0].Detailed.element_data[1].result_measurement := 0.00016298145, [0].Detailed.element_data[2].Variable_code := 13, [0].Detailed.element_data[2].prec_code := 3, [0].Detailed.element_data[2].Unit_code := 12, [0].Detailed.element_data[2].result_measurement := 5.1391406, [0].Detailed.element_data[3].Variable_code := 75, [0].Detailed.element_data[3].prec_code := 2, [0].Detailed.element_data[3].Unit_code := 60, [0].Detailed.element_data[4].Variable_code := 60, [0].Detailed.element_data[4].prec_code := 2, [0].Detailed.element_data[4].Unit_code := 60, [0].Detailed.element_data[4].result_measurement := -0.07711351, [0].Detailed.element_data[5].Variable_code := 56, [0].Detailed.element_data[5].prec_code := 3, [0].Detailed.element_data[5].Unit_code := 41, [0].Detailed.element_data[5].result_measurement := 0.00014901161, [0].Detailed.element_data[6].Variable_code := 55, [0].Detailed.element_data[6].prec_code := 3, [0].Detailed.element_data[6].Unit_code := 12, [0].Detailed.element_data[6].result_measurement := 5.1391406, [0].Detailed.element_data[7].Variable_code := 58, [0].Detailed.element_data[7].prec_code := 2, [0].Detailed.element_data[7].Unit_code := 60, [0].Detailed.element_data[7].result_measurement := -1.0002404, [0].Detailed.element_data[8].Variable_code := 59, [0].Detailed.element_data[8].prec_code := 2, [0].Detailed.element_data[8].Unit_code := 60, [0].Detailed.element_data[8].result_measurement := 1.0002404, [0].Detailed.element_data[9].Variable_code := 12, [0].Detailed.element_data[9].prec_code := 3, [0].Detailed.element_data[9].Unit_code := 12, [0].Detailed.element_data[9].result_measurement := 5.000001, [0].Detailed.element_data[10].Variable_code := 62,
        [0].Detailed.element_data[10].prec_code := 2, [0].Detailed.element_data[10].Unit_code := 60, [0].Detailed.element_data[10].result_measurement := 1.1002644, [0].Detailed.element_data[11].Variable_code := 21, [0].Detailed.element_data[11].prec_code := 3, [0].Detailed.element_data[11].Unit_code := 41, [0].Detailed.element_data[11].result_measurement := 0.0015180558, [0].Detailed.element_data[12].Variable_code := 25, [0].Detailed.element_data[12].prec_code := 3, [0].Detailed.element_data[12].Unit_code := 41, [0].Detailed.element_data[12].result_measurement := 0.021727756, [0].Detailed.element_data[13].Variable_code := 216, [0].Detailed.element_data[13].prec_code := 3, [0].Detailed.element_data[13].Unit_code := 41, [0].Detailed.element_data[13].result_measurement := 0.00085681677, [0].Detailed.element_data[14].Variable_code := 218, [0].Detailed.element_data[14].prec_code := 3, [0].Detailed.element_data[14].Unit_code := 41, [0].Detailed.element_data[14].result_measurement := 0.01094304, [0].Detailed.element_data[15].Variable_code := 295, [0].Detailed.element_data[15].prec_code := 3, [0].Detailed.element_data[15].Unit_code := 12, [0].Detailed.element_data[15].result_measurement := 5.140961, [1].UID := 41956, [1].Basic.unique_id := 41956, [1].Basic.channel_num := 1, [1].Basic.program_num := 2, [1].Basic.evaluation_code := 1, [1].Basic.test_port := 1, [1].Basic.year := 26, [1].Basic.month := 6, [1].Basic.date := 4, [1].Basic.hour := 14, [1].Basic.minute := 58, [1].Basic.second := 25, [1].Basic.flags := 12, [1].Basic.Num_tests := 1, [1].Basic.test_elements.test_type := 66, [1].Basic.test_elements.test_eval := 1, [1].Basic.test_elements.num_elements := 16, [1].Detailed.unique_id := 41956, [1].Detailed.num_elements := 16, [1].Detailed.Test_Type := 66, [1].Detailed.element_data[0].Variable_code := 61, [1].Detailed.element_data[0].prec_code := 2, [1].Detailed.element_data[0].Unit_code := 60, [1].Detailed.element_data[0].result_measurement := -0.06984919, [1].Detailed.element_data[1].Variable_code := 28, [1].Detailed.element_data[1].prec_code := 3, [1].Detailed.element_data[1].Unit_code := 41, [1].Detailed.element_data[1].result_measurement := 0.00022817403, [1].Detailed.element_data[2].Variable_code := 13, [1].Detailed.element_data[2].prec_code := 3, [1].Detailed.element_data[2].Unit_code := 12, [1].Detailed.element_data[2].result_measurement := 5.137343, [1].Detailed.element_data[3].Variable_code := 75, [1].Detailed.element_data[3].prec_code := 2, [1].Detailed.element_data[3].Unit_code := 60, [1].Detailed.element_data[4].Variable_code := 60, [1].Detailed.element_data[4].prec_code := 2,
        [1].Detailed.element_data[4].Unit_code := 60, [1].Detailed.element_data[4].result_measurement := -0.07878989, [1].Detailed.element_data[5].Variable_code := 56, [1].Detailed.element_data[5].prec_code := 3, [1].Detailed.element_data[5].Unit_code := 41, [1].Detailed.element_data[5].result_measurement := 0.00013038516, [1].Detailed.element_data[6].Variable_code := 55, [1].Detailed.element_data[6].prec_code := 3, [1].Detailed.element_data[6].Unit_code := 12, [1].Detailed.element_data[6].result_measurement := 5.137343, [1].Detailed.element_data[7].Variable_code := 58, [1].Detailed.element_data[7].prec_code := 2, [1].Detailed.element_data[7].Unit_code := 60, [1].Detailed.element_data[7].result_measurement := -1.0002404, [1].Detailed.element_data[8].Variable_code := 59, [1].Detailed.element_data[8].prec_code := 2, [1].Detailed.element_data[8].Unit_code := 60, [1].Detailed.element_data[8].result_measurement := 1.0002404, [1].Detailed.element_data[9].Variable_code := 12, [1].Detailed.element_data[9].prec_code := 3, [1].Detailed.element_data[9].Unit_code := 12, [1].Detailed.element_data[9].result_measurement := 5.000001, [1].Detailed.element_data[10].Variable_code := 62, [1].Detailed.element_data[10].prec_code := 2, [1].Detailed.element_data[10].Unit_code := 60, [1].Detailed.element_data[10].result_measurement := 1.1002644, [1].Detailed.element_data[11].Variable_code := 21, [1].Detailed.element_data[11].prec_code := 3, [1].Detailed.element_data[11].Unit_code := 41, [1].Detailed.element_data[11].result_measurement := 0.0015180558, [1].Detailed.element_data[12].Variable_code := 25, [1].Detailed.element_data[12].prec_code := 3, [1].Detailed.element_data[12].Unit_code := 41, [1].Detailed.element_data[12].result_measurement := 0.021727756, [1].Detailed.element_data[13].Variable_code := 216, [1].Detailed.element_data[13].prec_code := 3, [1].Detailed.element_data[13].Unit_code := 41, [1].Detailed.element_data[13].result_measurement := 0.00085681677, [1].Detailed.element_data[14].Variable_code := 218, [1].Detailed.element_data[14].prec_code := 3, [1].Detailed.element_data[14].Unit_code := 41, [1].Detailed.element_data[14].result_measurement := 0.01094304, [1].Detailed.element_data[15].Variable_code := 295, [1].Detailed.element_data[15].prec_code := 3, [1].Detailed.element_data[15].Unit_code := 12, [1].Detailed.element_data[15].result_measurement := 5.1386003, [2].UID := 41959, [2].Basic.unique_id := 41959, [2].Basic.channel_num := 1, [2].Basic.program_num := 2, [2].Basic.evaluation_code := 1, [2].Basic.test_port := 1, [2].Basic.year := 26, [2].Basic.month := 6, [2].Basic.date := 4, [2].Basic.hour := 15, [2].Basic.minute := 3, [2].Basic.second := 17, [2].Basic.flags := 12, [2].Basic.Num_tests := 1,
        [2].Basic.test_elements.test_type := 66, [2].Basic.test_elements.test_eval := 1, [2].Basic.test_elements.num_elements := 16, [2].Detailed.unique_id := 41959, [2].Detailed.num_elements := 16, [2].Detailed.Test_Type := 66, [2].Detailed.element_data[0].Variable_code := 61, [2].Detailed.element_data[0].prec_code := 2, [2].Detailed.element_data[0].Unit_code := 60, [2].Detailed.element_data[0].result_measurement := -0.06258488, [2].Detailed.element_data[1].Variable_code := 28, [2].Detailed.element_data[1].prec_code := 3, [2].Detailed.element_data[1].Unit_code := 41, [2].Detailed.element_data[1].result_measurement := 0.00036787242, [2].Detailed.element_data[2].Variable_code := 13, [2].Detailed.element_data[2].prec_code := 3, [2].Detailed.element_data[2].Unit_code := 12, [2].Detailed.element_data[2].result_measurement := 5.1356993, [2].Detailed.element_data[3].Variable_code := 75, [2].Detailed.element_data[3].prec_code := 2, [2].Detailed.element_data[3].Unit_code := 60, [2].Detailed.element_data[4].Variable_code := 60, [2].Detailed.element_data[4].prec_code := 2, [2].Detailed.element_data[4].Unit_code := 60, [2].Detailed.element_data[4].result_measurement := -0.073201954, [2].Detailed.element_data[5].Variable_code := 56, [2].Detailed.element_data[5].prec_code := 3, [2].Detailed.element_data[5].Unit_code := 41, [2].Detailed.element_data[5].result_measurement := 0.0001816079, [2].Detailed.element_data[6].Variable_code := 55, [2].Detailed.element_data[6].prec_code := 3, [2].Detailed.element_data[6].Unit_code := 12, [2].Detailed.element_data[6].result_measurement := 5.1356993, [2].Detailed.element_data[7].Variable_code := 58, [2].Detailed.element_data[7].prec_code := 2, [2].Detailed.element_data[7].Unit_code := 60, [2].Detailed.element_data[7].result_measurement := -1.0002404, [2].Detailed.element_data[8].Variable_code := 59, [2].Detailed.element_data[8].prec_code := 2, [2].Detailed.element_data[8].Unit_code := 60, [2].Detailed.element_data[8].result_measurement := 1.0002404, [2].Detailed.element_data[9].Variable_code := 12, [2].Detailed.element_data[9].prec_code := 3, [2].Detailed.element_data[9].Unit_code := 12, [2].Detailed.element_data[9].result_measurement := 5.000001, [2].Detailed.element_data[10].Variable_code := 62, [2].Detailed.element_data[10].prec_code := 2, [2].Detailed.element_data[10].Unit_code := 60, [2].Detailed.element_data[10].result_measurement := 1.1002644, [2].Detailed.element_data[11].Variable_code := 21, [2].Detailed.element_data[11].prec_code := 3, [2].Detailed.element_data[11].Unit_code := 41, [2].Detailed.element_data[11].result_measurement := 0.0015180558, [2].Detailed.element_data[12].Variable_code := 25, [2].Detailed.element_data[12].prec_code := 3, [2].Detailed.element_data[12].Unit_code := 41, [2].Detailed.element_data[12].result_measurement := 0.021727756, [2].Detailed.element_data[13].Variable_code := 216, [2].Detailed.element_data[13].prec_code := 3, [2].Detailed.element_data[13].Unit_code := 41,
        [2].Detailed.element_data[13].result_measurement := 0.00085681677, [2].Detailed.element_data[14].Variable_code := 218, [2].Detailed.element_data[14].prec_code := 3, [2].Detailed.element_data[14].Unit_code := 41, [2].Detailed.element_data[14].result_measurement := 0.01094304, [2].Detailed.element_data[15].Variable_code := 295, [2].Detailed.element_data[15].prec_code := 3, [2].Detailed.element_data[15].Unit_code := 12, [2].Detailed.element_data[15].result_measurement := 5.1374407, [3].UID := 41962, [3].Basic.unique_id := 41962, [3].Basic.channel_num := 1, [3].Basic.program_num := 2, [3].Basic.evaluation_code := 1, [3].Basic.test_port := 1, [3].Basic.year := 26, [3].Basic.month := 6, [3].Basic.date := 4, [3].Basic.hour := 15, [3].Basic.minute := 6, [3].Basic.second := 39, [3].Basic.flags := 12, [3].Basic.Num_tests := 1, [3].Basic.test_elements.test_type := 66, [3].Basic.test_elements.test_eval := 1, [3].Basic.test_elements.num_elements := 16, [3].Detailed.unique_id := 41962, [3].Detailed.num_elements := 16, [3].Detailed.Test_Type := 66, [3].Detailed.element_data[0].Variable_code := 61, [3].Detailed.element_data[0].prec_code := 2, [3].Detailed.element_data[0].Unit_code := 60, [3].Detailed.element_data[0].result_measurement := -0.058673322, [3].Detailed.element_data[1].Variable_code := 28, [3].Detailed.element_data[1].prec_code := 3, [3].Detailed.element_data[1].Unit_code := 41, [3].Detailed.element_data[1].result_measurement := 0.000433065, [3].Detailed.element_data[2].Variable_code := 13, [3].Detailed.element_data[2].prec_code := 3, [3].Detailed.element_data[2].Unit_code := 12, [3].Detailed.element_data[2].result_measurement := 5.136598, [3].Detailed.element_data[3].Variable_code := 75, [3].Detailed.element_data[3].prec_code := 2, [3].Detailed.element_data[3].Unit_code := 60, [3].Detailed.element_data[4].Variable_code := 60, [3].Detailed.element_data[4].prec_code := 2, [3].Detailed.element_data[4].Unit_code := 60, [3].Detailed.element_data[4].result_measurement := -0.06649643, [3].Detailed.element_data[5].Variable_code := 56, [3].Detailed.element_data[5].prec_code := 3, [3].Detailed.element_data[5].Unit_code := 41, [3].Detailed.element_data[5].result_measurement := 0.00024214387, [3].Detailed.element_data[6].Variable_code := 55, [3].Detailed.element_data[6].prec_code := 3, [3].Detailed.element_data[6].Unit_code := 12, [3].Detailed.element_data[6].result_measurement := 5.136598, [3].Detailed.element_data[7].Variable_code := 58, [3].Detailed.element_data[7].prec_code := 2, [3].Detailed.element_data[7].Unit_code := 60, [3].Detailed.element_data[7].result_measurement := -1.0002404,
